KUKA KRL program: EPS_2_25862_MH01_A_20251016040654.src

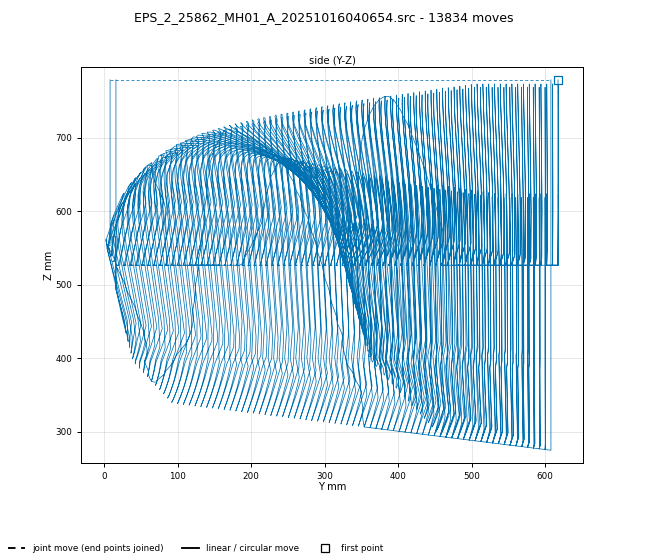
[picture p0: tool path of EPS_2_25862_MH01_A_20251016040654.src, 13834 of 13836 moves have a stored position in this frame; points joined in program order, loops and branches not executed]
&ACCESS RVP
&REL 4
&COMMENT QRS 19112012
&PARAM EDITMASK = *
DEF PART()
EXT BAS (BAS_COMMAND :IN,REAL :IN )
INT I
BAS (#INITMOV,0 )

;KUKA QRS Post kuka4.cps  Date:22-06-2017 !

File_ID=2893

QRS_PRE_INIT()

;Init var - Until changes are made in qrs_pre_init
Outlet_Square_prg=0
Inlet_1_Square_prg=0
Inlet_2_Square_prg=0
Inlet_3_Square_prg=0
Inlet_4_Square_prg=0
Inlet_5_Square_prg=0

Outlet_1={X 0.000, Y 506.950, Z 586.000, B 0.000, E1 0.000 }
Inlet_1={X 0.000, Y 532.640, Z 498.500, B 0.000, E1 270.000 }
Outlet_1_type=366
Inlet_1_type=201
;QRS#1=Sidecore dimensions
;QRS#2=375-15" PVC SDR 35
;QRS#3=200-8" PVC SDR 35
;QRS#4=
;QRS#5=
;QRS#6=
;QRS#7=
;QRS#8=
;QRS#9=20Y PSX
;QRS#10=12-08 PSX
;QRS#11=
;QRS#12=
;QRS#13=
;QRS#14=
;QRS#15=
;QRS#16=1220x127x1067 3,5'
;QRS#17=EPS Height
;QRS#18=769
;QRS#19=*
;QRS#20= UPDATED VERSION 22-06-2017
;QRS#21=*
Outlet_Square=0250
Inlet_1_Square=0100
Inlet_2_Square=0
Inlet_3_Square=0
Inlet_4_Square=0
Inlet_5_Square=0
Mill_Square=1
Outlet_Square_Prg=252
Inlet_1_Square_prg=204

QRS_INIT()

$ADVANCE=5

; T1
PTP {E1 171.211,E2 171.211}
PTP {X 0,Y 617.567,A -85,B 0,C 180,E1 171.211,E2 171.211,E3 0,E4 0,E5 0,E6 0}
QRS_SPEED_INIT()
LIN {X 0,Y 617.567,Z 779,A -85,B 0,C 180,E1 171.211,E2 171.211,E3 0,E4 0,E5 0,E6 0} C_VEL
LIN {X 0,Y 617.567,Z 528.81,A -85,B 0,C 180,E1 171.211,E2 171.211} C_VEL
LIN {X 0,Y 617.544,Z 526.81,A -85,B 0,C 180,E1 171.397,E2 171.397} C_VEL
LIN {X 0,Y 617.991,Z 526.81,A -85,B 0,C 180,E1 174.215,E2 174.215} C_VEL
LIN {X 0,Y 618.006,Z 526.81,A -85,B 0,C 180,E1 178.846,E2 178.846} C_VEL
LIN {X 0,Y 618.053,Z 526.81,A -85,B 0,C 180,E1 183.469,E2 183.469} C_VEL
LIN {X 0,Y 617.988,Z 526.81,A -85,B 0,C 180,E1 188.116,E2 188.116} C_VEL
LIN {X 0,Y 617.951,Z 526.81,A -85,B 0,C 180,E1 192.817,E2 192.817} C_VEL
LIN {X 0,Y 617.958,Z 526.81,A -85,B 0,C 180,E1 197.608,E2 197.608} C_VEL
LIN {X 0,Y 617.766,Z 526.81,A -85,B 0,C 180,E1 198.549,E2 198.549} C_VEL
LIN {X 0,Y 617.884,Z 526.81,A -85,B 0,C 180,E1 202.532,E2 202.532} C_VEL
LIN {X 0,Y 617.406,Z 526.81,A -85,B 0,C 180,E1 205.079,E2 205.079} C_VEL
LIN {X 0,Y 617.875,Z 526.81,A -85,B 0,C 180,E1 207.638,E2 207.638} C_VEL
LIN {X 0,Y 617.419,Z 526.81,A -85,B 0,C 180,E1 210.304,E2 210.304} C_VEL
LIN {X 0,Y 617.937,Z 526.81,A -85,B 0,C 180,E1 212.99,E2 212.99} C_VEL
LIN {X 0,Y 617.675,Z 526.81,A -85,B 0,C 180,E1 215.809,E2 215.809} C_VEL
LIN {X 0,Y 617.669,Z 526.81,A -85,B 0,C 180,E1 218.112,E2 218.112} C_VEL
LIN {X 0,Y 617.756,Z 526.81,A -85,B 0,C 180,E1 221.735,E2 221.735} C_VEL
LIN {X 0,Y 617.383,Z 526.81,A -85,B 0,C 180,E1 225.055,E2 225.055} C_VEL
LIN {X 0,Y 617.751,Z 526.81,A -85,B 0,C 180,E1 228.278,E2 228.278} C_VEL
LIN {X 0,Y 617.353,Z 526.81,A -85,B 0,C 180,E1 231.927,E2 231.927} C_VEL
LIN {X 0,Y 617.814,Z 526.81,A -85,B 0,C 180,E1 234.203,E2 234.203} C_VEL
LIN {X 0,Y 617.316,Z 526.81,A -85,B 0,C 180,E1 236.974,E2 236.974} C_VEL
LIN {X 0,Y 617.844,Z 526.81,A -85,B 0,C 180,E1 239.721,E2 239.721} C_VEL
LIN {X 0,Y 617.407,Z 526.81,A -85,B 0,C 180,E1 242.341,E2 242.341} C_VEL
LIN {X 0,Y 617.943,Z 526.81,A -85,B 0,C 180,E1 244.946,E2 244.946} C_VEL
LIN {X 0,Y 618.003,Z 526.81,A -85,B 0,C 180,E1 249.132,E2 249.132} C_VEL
LIN {X 0,Y 617.672,Z 526.81,A -85,B 0,C 180,E1 249.232,E2 249.232} C_VEL
LIN {X 0,Y 617.573,Z 527.124,A -85,B 0,C 180,E1 249.254,E2 249.254} C_VEL
LIN {X 0,Y 617.998,Z 591.592,A -85,B 0,C 180,E1 250.062,E2 250.062} C_VEL
LIN {X 0,Y 618.002,Z 600.715,A -85,B 0,C 180,E1 250.212,E2 250.212} C_VEL
LIN {X 0,Y 617.91,Z 609.031,A -85,B 0,C 180,E1 250.381,E2 250.381} C_VEL
LIN {X 0,Y 617.97,Z 618.416,A -85,B 0,C 180,E1 250.619,E2 250.619} C_VEL
LIN {X 0,Y 617.998,Z 627.724,A -85,B 0,C 180,E1 250.899,E2 250.899} C_VEL
LIN {X 0,Y 617.96,Z 636.377,A -85,B 0,C 180,E1 251.197,E2 251.197} C_VEL
LIN {X 0,Y 617.966,Z 645.125,A -85,B 0,C 180,E1 251.542,E2 251.542} C_VEL
LIN {X 0,Y 618.001,Z 654.313,A -85,B 0,C 180,E1 251.955,E2 251.955} C_VEL
LIN {X 0,Y 617.987,Z 663.052,A -85,B 0,C 180,E1 252.395,E2 252.395} C_VEL
LIN {X 0,Y 617.974,Z 670.423,A -85,B 0,C 180,E1 252.803,E2 252.803} C_VEL
LIN {X 0,Y 617.99,Z 678.723,A -85,B 0,C 180,E1 253.313,E2 253.313} C_VEL
LIN {X 0,Y 617.989,Z 687.493,A -85,B 0,C 180,E1 253.911,E2 253.911} C_VEL
LIN {X 0,Y 617.973,Z 695.458,A -85,B 0,C 180,E1 254.511,E2 254.511} C_VEL
LIN {X 0,Y 617.955,Z 702.634,A -85,B 0,C 180,E1 255.102,E2 255.102} C_VEL
LIN {X 0,Y 617.942,Z 709.277,A -85,B 0,C 180,E1 255.699,E2 255.699} C_VEL
LIN {X 0,Y 617.983,Z 715.369,A -85,B 0,C 180,E1 256.295,E2 256.295} C_VEL
LIN {X 0,Y 617.985,Z 720.995,A -85,B 0,C 180,E1 256.889,E2 256.889} C_VEL
LIN {X 0,Y 617.92,Z 727.418,A -85,B 0,C 180,E1 257.628,E2 257.628} C_VEL
LIN {X 0,Y 617.926,Z 733.244,A -85,B 0,C 180,E1 258.366,E2 258.366} C_VEL
LIN {X 0,Y 617.973,Z 737.547,A -85,B 0,C 180,E1 258.956,E2 258.956} C_VEL
LIN {X 0,Y 617.979,Z 742.76,A -85,B 0,C 180,E1 259.742,E2 259.742} C_VEL
LIN {X 0,Y 617.882,Z 748.578,A -85,B 0,C 180,E1 260.724,E2 260.724} C_VEL
LIN {X 0,Y 617.911,Z 752.668,A -85,B 0,C 180,E1 261.501,E2 261.501} C_VEL
LIN {X 0,Y 618.002,Z 756.64,A -85,B 0,C 180,E1 262.353,E2 262.353} C_VEL
LIN {X 0,Y 617.904,Z 760.475,A -85,B 0,C 180,E1 263.283,E2 263.283} C_VEL
LIN {X 0,Y 617.879,Z 762.222,A -85,B 0,C 180,E1 263.748,E2 263.748} C_VEL
LIN {X 0,Y 617.937,Z 765.214,A -85,B 0,C 180,E1 264.678,E2 264.678} C_VEL
LIN {X 0,Y 617.962,Z 767.691,A -85,B 0,C 180,E1 265.606,E2 265.606} C_VEL
LIN {X 0,Y 617.845,Z 769.703,A -85,B 0,C 180,E1 266.532,E2 266.532} C_VEL
LIN {X 0,Y 617.849,Z 771.199,A -85,B 0,C 180,E1 267.457,E2 267.457} C_VEL
LIN {X 0,Y 617.951,Z 772.526,A -85,B 0,C 180,E1 268.845,E2 268.845} C_VEL
LIN {X 0,Y 617.842,Z 772.907,A -85,B 0,C 180,E1 269.769,E2 269.769} C_VEL
LIN {X 0,Y 617.828,Z 772.91,A -85,B 0,C 180,E1 270.232,E2 270.232} C_VEL
LIN {X 0,Y 617.89,Z 772.542,A -85,B 0,C 180,E1 271.156,E2 271.156} C_VEL
LIN {X 0,Y 617.878,Z 771.19,A -85,B 0,C 180,E1 272.544,E2 272.544} C_VEL
LIN {X 0,Y 617.83,Z 769.706,A -85,B 0,C 180,E1 273.47,E2 273.47} C_VEL
LIN {X 0,Y 617.92,Z 767.699,A -85,B 0,C 180,E1 274.396,E2 274.396} C_VEL
LIN {X 0,Y 617.979,Z 765.199,A -85,B 0,C 180,E1 275.323,E2 275.323} C_VEL
LIN {X 0,Y 617.884,Z 762.216,A -85,B 0,C 180,E1 276.253,E2 276.253} C_VEL
LIN {X 0,Y 617.945,Z 757.648,A -85,B 0,C 180,E1 277.416,E2 277.416} C_VEL
LIN {X 0,Y 617.97,Z 754.519,A -85,B 0,C 180,E1 278.115,E2 278.115} C_VEL
LIN {X 0,Y 617.888,Z 749.593,A -85,B 0,C 180,E1 279.09,E2 279.09} C_VEL
LIN {X 0,Y 617.902,Z 745.133,A -85,B 0,C 180,E1 279.871,E2 279.871} C_VEL
LIN {X 0,Y 617.972,Z 741.485,A -85,B 0,C 180,E1 280.457,E2 280.457} C_VEL
LIN {X 0,Y 617.979,Z 735.404,A -85,B 0,C 180,E1 281.339,E2 281.339} C_VEL
LIN {X 0,Y 617.924,Z 729.803,A -85,B 0,C 180,E1 282.078,E2 282.078} C_VEL
LIN {X 0,Y 617.94,Z 723.617,A -85,B 0,C 180,E1 282.817,E2 282.817} C_VEL
LIN {X 0,Y 618.001,Z 718.223,A -85,B 0,C 180,E1 283.409,E2 283.409} C_VEL
LIN {X 0,Y 617.984,Z 710.825,A -85,B 0,C 180,E1 284.152,E2 284.152} C_VEL
LIN {X 0,Y 617.966,Z 704.331,A -85,B 0,C 180,E1 284.749,E2 284.749} C_VEL
LIN {X 0,Y 617.984,Z 696.644,A -85,B 0,C 180,E1 285.394,E2 285.394} C_VEL
LIN {X 0,Y 617.986,Z 690.265,A -85,B 0,C 180,E1 285.886,E2 285.886} C_VEL
LIN {X 0,Y 618,Z 681.693,A -85,B 0,C 180,E1 286.489,E2 286.489} C_VEL
LIN {X 0,Y 617.987,Z 673.739,A -85,B 0,C 180,E1 286.996,E2 286.996} C_VEL
LIN {X 0,Y 617.97,Z 664.896,A -85,B 0,C 180,E1 287.505,E2 287.505} C_VEL
LIN {X 0,Y 617.953,Z 657.854,A -85,B 0,C 180,E1 287.873,E2 287.873} C_VEL
LIN {X 0,Y 617.995,Z 649.403,A -85,B 0,C 180,E1 288.27,E2 288.27} C_VEL
LIN {X 0,Y 617.999,Z 641.397,A -85,B 0,C 180,E1 288.609,E2 288.609} C_VEL
LIN {X 0,Y 617.905,Z 631.678,A -85,B 0,C 180,E1 288.973,E2 288.973} C_VEL
LIN {X 0,Y 618.012,Z 622.258,A -85,B 0,C 180,E1 289.27,E2 289.27} C_VEL
LIN {X 0,Y 618.03,Z 612.701,A -85,B 0,C 180,E1 289.528,E2 289.528} C_VEL
LIN {X 0,Y 617.968,Z 602.985,A -85,B 0,C 180,E1 289.746,E2 289.746} C_VEL
LIN {X 0,Y 617.848,Z 594.545,A -85,B 0,C 180,E1 289.901,E2 289.901} C_VEL
LIN {X 0,Y 617.823,Z 577.609,A -85,B 0,C 180,E1 290.124,E2 290.124} C_VEL
LIN {X 0,Y 617.563,Z 526.827,A -85,B 0,C 180,E1 290.75,E2 290.75} C_VEL
LIN {X 0,Y 618.055,Z 526.81,A -85,B 0,C 180,E1 290.891,E2 290.891} C_VEL
LIN {X 0,Y 617.945,Z 526.81,A -85,B 0,C 180,E1 295.055,E2 295.055} C_VEL
LIN {X 0,Y 617.401,Z 526.81,A -85,B 0,C 180,E1 297.66,E2 297.66} C_VEL
LIN {X 0,Y 617.83,Z 526.81,A -85,B 0,C 180,E1 300.281,E2 300.281} C_VEL
LIN {X 0,Y 617.31,Z 526.81,A -85,B 0,C 180,E1 303.028,E2 303.028} C_VEL
LIN {X 0,Y 617.818,Z 526.81,A -85,B 0,C 180,E1 305.798,E2 305.798} C_VEL
LIN {X 0,Y 617.553,Z 526.81,A -85,B 0,C 180,E1 308.722,E2 308.722} C_VEL
LIN {X 0,Y 617.772,Z 526.81,A -85,B 0,C 180,E1 311.733,E2 311.733} C_VEL
LIN {X 0,Y 617.89,Z 526.81,A -85,B 0,C 180,E1 315.1,E2 315.1} C_VEL
LIN {X 0,Y 617.463,Z 526.81,A -85,B 0,C 180,E1 318.307,E2 318.307} C_VEL
LIN {X 0,Y 617.793,Z 526.81,A -85,B 0,C 180,E1 321.295,E2 321.295} C_VEL
LIN {X 0,Y 617.729,Z 526.81,A -85,B 0,C 180,E1 325.801,E2 325.801} C_VEL
LIN {X 0,Y 617.882,Z 526.81,A -85,B 0,C 180,E1 327.006,E2 327.006} C_VEL
LIN {X 0,Y 617.635,Z 526.81,A -85,B 0,C 180,E1 330.177,E2 330.177} C_VEL
LIN {X 0,Y 617.646,Z 526.81,A -85,B 0,C 180,E1 332.351,E2 332.351} C_VEL
LIN {X 0,Y 617.512,Z 526.81,A -85,B 0,C 180,E1 335.244,E2 335.244} C_VEL
LIN {X 0,Y 617.731,Z 526.81,A -85,B 0,C 180,E1 337.462,E2 337.462} C_VEL
LIN {X 0,Y 617.771,Z 526.81,A -85,B 0,C 180,E1 341.453,E2 341.453} C_VEL
LIN {X 0,Y 617.968,Z 526.81,A -85,B 0,C 180,E1 342.392,E2 342.392} C_VEL
LIN {X 0,Y 617.72,Z 526.81,A -85,B 0,C 180,E1 347.178,E2 347.178} C_VEL
LIN {X 0,Y 617.945,Z 526.81,A -85,B 0,C 180,E1 348.034,E2 348.034} C_VEL
LIN {X 0,Y 617.433,Z 526.895,A -85,B 0,C 180,E1 348.173,E2 348.173} C_VEL
LIN {X 0,Y 617.979,Z 531.008,A -85,B 0,C 180,E1 348.301,E2 348.301} C_VEL
LIN {X 0,Y 617.99,Z 539.274,A -85,B 0,C 180,E1 348.568,E2 348.568} C_VEL
LIN {X 0,Y 618.035,Z 547.303,A -85,B 0,C 180,E1 348.887,E2 348.887} C_VEL
LIN {X 0,Y 618.042,Z 554.943,A -85,B 0,C 180,E1 349.245,E2 349.245} C_VEL
LIN {X 0,Y 617.989,Z 563.583,A -85,B 0,C 180,E1 349.726,E2 349.726} C_VEL
LIN {X 0,Y 618.017,Z 570.585,A -85,B 0,C 180,E1 350.186,E2 350.186} C_VEL
LIN {X 0,Y 618.022,Z 577.883,A -85,B 0,C 180,E1 350.735,E2 350.735} C_VEL
LIN {X 0,Y 617.995,Z 584.768,A -85,B 0,C 180,E1 351.337,E2 351.337} C_VEL
LIN {X 0,Y 617.992,Z 591.346,A -85,B 0,C 180,E1 352.001,E2 352.001} C_VEL
LIN {X 0,Y 617.99,Z 596.368,A -85,B 0,C 180,E1 352.584,E2 352.584} C_VEL
LIN {X 0,Y 617.999,Z 601.64,A -85,B 0,C 180,E1 353.282,E2 353.282} C_VEL
LIN {X 0,Y 617.979,Z 606.155,A -85,B 0,C 180,E1 353.98,E2 353.98} C_VEL
LIN {X 0,Y 617.965,Z 610.06,A -85,B 0,C 180,E1 354.676,E2 354.676} C_VEL
LIN {X 0,Y 618.005,Z 613.315,A -85,B 0,C 180,E1 355.372,E2 355.372} C_VEL
LIN {X 0,Y 617.99,Z 616.083,A -85,B 0,C 180,E1 356.067,E2 356.067} C_VEL
LIN {X 0,Y 617.961,Z 617.642,A -85,B 0,C 180,E1 356.53,E2 356.53} C_VEL
LIN {X 0,Y 617.962,Z 618.985,A -85,B 0,C 180,E1 356.993,E2 356.993} C_VEL
LIN {X 0,Y 617.986,Z 620.121,A -85,B 0,C 180,E1 357.456,E2 357.456} C_VEL
LIN {X 0,Y 617.984,Z 621.822,A -85,B 0,C 180,E1 358.381,E2 358.381} C_VEL
LIN {X 0,Y 617.941,Z 622.381,A -85,B 0,C 180,E1 358.843,E2 358.843} C_VEL
LIN {X 0,Y 617.943,Z 622.891,A -85,B 0,C 180,E1 359.767,E2 359.767} C_VEL
LIN {X 0,Y 617.998,Z 622.65,A -85,B 0,C 180,E1 360.692,E2 360.692} C_VEL
LIN {X 0,Y 617.929,Z 621.709,A -85,B 0,C 180,E1 361.616,E2 361.616} C_VEL
LIN {X 0,Y 617.952,Z 619.943,A -85,B 0,C 180,E1 362.541,E2 362.541} C_VEL
LIN {X 0,Y 617.986,Z 617.357,A -85,B 0,C 180,E1 363.467,E2 363.467} C_VEL
LIN {X 0,Y 617.958,Z 615.767,A -85,B 0,C 180,E1 363.93,E2 363.93} C_VEL
LIN {X 0,Y 617.962,Z 612.953,A -85,B 0,C 180,E1 364.625,E2 364.625} C_VEL
LIN {X 0,Y 618.012,Z 609.592,A -85,B 0,C 180,E1 365.32,E2 365.32} C_VEL
LIN {X 0,Y 618.005,Z 605.617,A -85,B 0,C 180,E1 366.017,E2 366.017} C_VEL
LIN {X 0,Y 617.996,Z 601.043,A -85,B 0,C 180,E1 366.715,E2 366.715} C_VEL
LIN {X 0,Y 618.007,Z 595.651,A -85,B 0,C 180,E1 367.413,E2 367.413} C_VEL
LIN {X 0,Y 618.016,Z 589.425,A -85,B 0,C 180,E1 368.112,E2 368.112} C_VEL
LIN {X 0,Y 618.01,Z 582.569,A -85,B 0,C 180,E1 368.777,E2 368.777} C_VEL
LIN {X 0,Y 617.987,Z 575.788,A -85,B 0,C 180,E1 369.34,E2 369.34} C_VEL
LIN {X 0,Y 618.031,Z 568.063,A -85,B 0,C 180,E1 369.896,E2 369.896} C_VEL
LIN {X 0,Y 618.031,Z 560.563,A -85,B 0,C 180,E1 370.36,E2 370.36} C_VEL
LIN {X 0,Y 617.996,Z 552.876,A -85,B 0,C 180,E1 370.768,E2 370.768} C_VEL
LIN {X 0,Y 618.051,Z 545.241,A -85,B 0,C 180,E1 371.11,E2 371.11} C_VEL
LIN {X 0,Y 618.043,Z 537.066,A -85,B 0,C 180,E1 371.418,E2 371.418} C_VEL
LIN {X 0,Y 617.95,Z 527.367,A -85,B 0,C 180,E1 371.71,E2 371.71} C_VEL
LIN {X 0,Y 617.836,Z 526.81,A -85,B 0,C 180,E1 371.732,E2 371.732} C_VEL
LIN {X 0,Y 618.049,Z 526.81,A -85,B 0,C 180,E1 371.961,E2 371.961} C_VEL
LIN {X 0,Y 617.965,Z 526.81,A -85,B 0,C 180,E1 377.604,E2 377.604} C_VEL
LIN {X 0,Y 617.784,Z 526.81,A -85,B 0,C 180,E1 378.551,E2 378.551} C_VEL
LIN {X 0,Y 617.94,Z 526.81,A -85,B 0,C 180,E1 382.527,E2 382.527} C_VEL
LIN {X 0,Y 617.438,Z 526.81,A -85,B 0,C 180,E1 385.074,E2 385.074} C_VEL
LIN {X 0,Y 617.879,Z 526.81,A -85,B 0,C 180,E1 387.634,E2 387.634} C_VEL
LIN {X 0,Y 617.37,Z 526.81,A -85,B 0,C 180,E1 390.303,E2 390.303} C_VEL
LIN {X 0,Y 617.844,Z 526.81,A -85,B 0,C 180,E1 392.992,E2 392.992} C_VEL
LIN {X 0,Y 617.702,Z 526.81,A -85,B 0,C 180,E1 394.195,E2 394.195} C_VEL
LIN {X 0,Y 617.786,Z 526.81,A -85,B 0,C 180,E1 398.701,E2 398.701} C_VEL
LIN {X 0,Y 617.438,Z 526.81,A -85,B 0,C 180,E1 401.757,E2 401.757} C_VEL
LIN {X 0,Y 617.869,Z 526.81,A -85,B 0,C 180,E1 404.898,E2 404.898} C_VEL
LIN {X 0,Y 617.794,Z 526.81,A -85,B 0,C 180,E1 408.269,E2 408.269} C_VEL
LIN {X 0,Y 617.56,Z 526.81,A -85,B 0,C 180,E1 411.279,E2 411.279} C_VEL
LIN {X 0,Y 617.58,Z 526.81,A -85,B 0,C 180,E1 411.896,E2 411.896} C_VEL
LIN {X 0,Y 617.811,Z 526.81,A -85,B 0,C 180,E1 414.201,E2 414.201} C_VEL
LIN {X 0,Y 617.354,Z 526.81,A -85,B 0,C 180,E1 416.975,E2 416.975} C_VEL
LIN {X 0,Y 617.897,Z 526.81,A -85,B 0,C 180,E1 419.722,E2 419.722} C_VEL
LIN {X 0,Y 617.42,Z 526.81,A -85,B 0,C 180,E1 422.341,E2 422.341} C_VEL
LIN {X 0,Y 617.901,Z 526.81,A -85,B 0,C 180,E1 424.943,E2 424.943} C_VEL
LIN {X 0,Y 617.445,Z 526.81,A -85,B 0,C 180,E1 427.451,E2 427.451} C_VEL
LIN {X 0,Y 617.945,Z 526.81,A -85,B 0,C 180,E1 429.951,E2 429.951} C_VEL
LIN {X 0,Y 618.027,Z 526.81,A -85,B 0,C 180,E1 433.628,E2 433.628} C_VEL
LIN {X 0,Y 618.006,Z 526.81,A -85,B 0,C 180,E1 439.544,E2 439.544} C_VEL
LIN {X 0,Y 618.005,Z 526.81,A -85,B 0,C 180,E1 444.213,E2 444.213} C_VEL
LIN {X 0,Y 618.056,Z 526.81,A -85,B 0,C 180,E1 448.844,E2 448.844} C_VEL
LIN {X 0,Y 618.059,Z 526.81,A -85,B 0,C 180,E1 453.467,E2 453.467} C_VEL
LIN {X 0,Y 617.996,Z 526.81,A -85,B 0,C 180,E1 458.114,E2 458.114} C_VEL
LIN {X 0,Y 618.005,Z 526.81,A -85,B 0,C 180,E1 462.814,E2 462.814} C_VEL
LIN {X 0,Y 617.945,Z 526.81,A -85,B 0,C 180,E1 467.606,E2 467.606} C_VEL
LIN {X 0,Y 617.762,Z 526.81,A -85,B 0,C 180,E1 468.554,E2 468.554} C_VEL
LIN {X 0,Y 617.921,Z 526.81,A -85,B 0,C 180,E1 472.529,E2 472.529} C_VEL
LIN {X 0,Y 617.422,Z 526.81,A -85,B 0,C 180,E1 475.076,E2 475.076} C_VEL
LIN {X 0,Y 617.864,Z 526.81,A -85,B 0,C 180,E1 477.637,E2 477.637} C_VEL
LIN {X 0,Y 617.365,Z 526.81,A -85,B 0,C 180,E1 480.305,E2 480.305} C_VEL
LIN {X 0,Y 617.849,Z 526.81,A -85,B 0,C 180,E1 482.994,E2 482.994} C_VEL
LIN {X 0,Y 617.717,Z 526.81,A -85,B 0,C 180,E1 484.202,E2 484.202} C_VEL
LIN {X 0,Y 617.776,Z 526.81,A -85,B 0,C 180,E1 488.704,E2 488.704} C_VEL
LIN {X 0,Y 617.417,Z 526.81,A -85,B 0,C 180,E1 491.761,E2 491.761} C_VEL
LIN {X 0,Y 617.82,Z 526.81,A -85,B 0,C 180,E1 494.905,E2 494.905} C_VEL
LIN {X 0,Y 617.766,Z 526.81,A -85,B 0,C 180,E1 498.274,E2 498.274} C_VEL
LIN {X 0,Y 617.556,Z 526.81,A -85,B 0,C 180,E1 501.282,E2 501.282} C_VEL
LIN {X 0,Y 617.832,Z 526.81,A -85,B 0,C 180,E1 504.206,E2 504.206} C_VEL
LIN {X 0,Y 617.356,Z 526.81,A -85,B 0,C 180,E1 506.978,E2 506.978} C_VEL
LIN {X 0,Y 617.899,Z 526.81,A -85,B 0,C 180,E1 509.725,E2 509.725} C_VEL
LIN {X 0,Y 617.405,Z 526.81,A -85,B 0,C 180,E1 512.343,E2 512.343} C_VEL
LIN {X 0,Y 617.874,Z 526.81,A -85,B 0,C 180,E1 514.945,E2 514.945} C_VEL
LIN {X 0,Y 617.444,Z 526.81,A -85,B 0,C 180,E1 517.454,E2 517.454} C_VEL
LIN {X 0,Y 617.969,Z 526.81,A -85,B 0,C 180,E1 519.954,E2 519.954} C_VEL
LIN {X 0,Y 618.057,Z 526.81,A -85,B 0,C 180,E1 523.625,E2 523.625} C_VEL
LIN {X 0,Y 618.006,Z 526.81,A -85,B 0,C 180,E1 529.546,E2 529.546} C_VEL
LIN {X 0,Y 617.544,Z 526.81,A -85,B 0,C 180,E1 531.397,E2 531.397} C_VEL
LIN {X 0,Y 613.845,Z 526.81,A -85,B 0,C 180,E1 532.988,E2 532.988} C_VEL
LIN {X 0,Y 609.944,Z 526.81,A -85,B 0,C 180,E1 534.598,E2 534.598} C_VEL
LIN {X 0,Y 609.767,Z 526.81,A -85,B 0,C 180,E1 539.996,E2 539.996} C_VEL
LIN {X 0,Y 609.877,Z 526.81,A -85,B 0,C 180,E1 544.267,E2 544.267} C_VEL
LIN {X 0,Y 609.912,Z 526.81,A -85,B 0,C 180,E1 548.561,E2 548.561} C_VEL
LIN {X 0,Y 610.024,Z 526.81,A -85,B 0,C 180,E1 552.902,E2 552.902} C_VEL
LIN {X 0,Y 609.801,Z 526.81,A -85,B 0,C 180,E1 558.825,E2 558.825} C_VEL
LIN {X 0,Y 609.689,Z 526.81,A -85,B 0,C 180,E1 563.406,E2 563.406} C_VEL
LIN {X 0,Y 609.802,Z 526.81,A -85,B 0,C 180,E1 568.141,E2 568.141} C_VEL
LIN {X 0,Y 610.014,Z 526.81,A -85,B 0,C 180,E1 573.089,E2 573.089} C_VEL
LIN {X 0,Y 609.701,Z 526.81,A -85,B 0,C 180,E1 578.368,E2 578.368} C_VEL
LIN {X 0,Y 609.712,Z 526.81,A -85,B 0,C 180,E1 582.095,E2 582.095} C_VEL
LIN {X 0,Y 609.791,Z 526.81,A -85,B 0,C 180,E1 588.139,E2 588.139} C_VEL
LIN {X 0,Y 609.673,Z 526.81,A -85,B 0,C 180,E1 593.419,E2 593.419} C_VEL
LIN {X 0,Y 609.781,Z 526.81,A -85,B 0,C 180,E1 600.229,E2 600.229} C_VEL
LIN {X 0,Y 610.026,Z 526.81,A -85,B 0,C 180,E1 605.047,E2 605.047} C_VEL
LIN {X 0,Y 610.064,Z 526.839,A -85,B 0,C 180,E1 608.983,E2 608.983} C_VEL
LIN {X 0,Y 610.516,Z 606.691,A -85,B 0,C 180,E1 610.077,E2 610.077} C_VEL
LIN {X 0,Y 610.436,Z 640.436,A -85,B 0,C 180,E1 611.114,E2 611.114} C_VEL
LIN {X 0,Y 610.334,Z 672.149,A -85,B 0,C 180,E1 612.685,E2 612.685} C_VEL
LIN {X 0,Y 610.259,Z 700.151,A -85,B 0,C 180,E1 614.678,E2 614.678} C_VEL
LIN {X 0,Y 610.211,Z 724.689,A -85,B 0,C 180,E1 617.1,E2 617.1} C_VEL
LIN {X 0,Y 610.176,Z 744.633,A -85,B 0,C 180,E1 619.82,E2 619.82} C_VEL
LIN {X 0,Y 610.138,Z 760.105,A -85,B 0,C 180,E1 622.876,E2 622.876} C_VEL
LIN {X 0,Y 610.138,Z 769.078,A -85,B 0,C 180,E1 625.734,E2 625.734} C_VEL
LIN {X 0,Y 610.097,Z 773.418,A -85,B 0,C 180,E1 628.581,E2 628.581} C_VEL
LIN {X 0,Y 610.054,Z 773.413,A -85,B 0,C 180,E1 631.426,E2 631.426} C_VEL
LIN {X 0,Y 610.083,Z 769.063,A -85,B 0,C 180,E1 634.273,E2 634.273} C_VEL
LIN {X 0,Y 610.151,Z 758.546,A -85,B 0,C 180,E1 637.489,E2 637.489} C_VEL
LIN {X 0,Y 610.185,Z 742.34,A -85,B 0,C 180,E1 640.548,E2 640.548} C_VEL
LIN {X 0,Y 610.211,Z 721.418,A -85,B 0,C 180,E1 643.272,E2 643.272} C_VEL
LIN {X 0,Y 610.288,Z 695.834,A -85,B 0,C 180,E1 645.67,E2 645.67} C_VEL
LIN {X 0,Y 610.359,Z 667.256,A -85,B 0,C 180,E1 647.601,E2 647.601} C_VEL
LIN {X 0,Y 610.454,Z 634.794,A -85,B 0,C 180,E1 649.105,E2 649.105} C_VEL
LIN {X 0,Y 610.49,Z 600.135,A -85,B 0,C 180,E1 650.053,E2 650.053} C_VEL
LIN {X 0,Y 610.11,Z 526.81,A -85,B 0,C 180,E1 651.046,E2 651.046} C_VEL
LIN {X 0,Y 610.033,Z 526.81,A -85,B 0,C 180,E1 654.96,E2 654.96} C_VEL
LIN {X 0,Y 609.762,Z 526.81,A -85,B 0,C 180,E1 659.78,E2 659.78} C_VEL
LIN {X 0,Y 609.718,Z 526.81,A -85,B 0,C 180,E1 666.586,E2 666.586} C_VEL
LIN {X 0,Y 609.78,Z 526.81,A -85,B 0,C 180,E1 672.103,E2 672.103} C_VEL
LIN {X 0,Y 609.523,Z 526.81,A -85,B 0,C 180,E1 677.889,E2 677.889} C_VEL
LIN {X 0,Y 609.488,Z 526.81,A -85,B 0,C 180,E1 682.654,E2 682.654} C_VEL
LIN {X 0,Y 609.824,Z 526.81,A -85,B 0,C 180,E1 687.587,E2 687.587} C_VEL
LIN {X 0,Y 609.683,Z 526.81,A -85,B 0,C 180,E1 691.853,E2 691.853} C_VEL
LIN {X 0,Y 609.663,Z 526.81,A -85,B 0,C 180,E1 696.771,E2 696.771} C_VEL
LIN {X 0,Y 609.947,Z 526.81,A -85,B 0,C 180,E1 702.675,E2 702.675} C_VEL
LIN {X 0,Y 609.764,Z 526.81,A -85,B 0,C 180,E1 708.003,E2 708.003} C_VEL
LIN {X 0,Y 610.311,Z 553.498,A -85,B 0,C 180,E1 709.011,E2 709.011} C_VEL
LIN {X 0,Y 610.246,Z 576.43,A -85,B 0,C 180,E1 710.454,E2 710.454} C_VEL
LIN {X 0,Y 610.193,Z 595.738,A -85,B 0,C 180,E1 712.32,E2 712.32} C_VEL
LIN {X 0,Y 610.161,Z 609.339,A -85,B 0,C 180,E1 714.308,E2 714.308} C_VEL
LIN {X 0,Y 610.141,Z 619.6,A -85,B 0,C 180,E1 716.804,E2 716.804} C_VEL
LIN {X 0,Y 610.148,Z 623.152,A -85,B 0,C 180,E1 718.583,E2 718.583} C_VEL
LIN {X 0,Y 610.156,Z 623.995,A -85,B 0,C 180,E1 720.004,E2 720.004} C_VEL
LIN {X 0,Y 610.126,Z 621.914,A -85,B 0,C 180,E1 722.138,E2 722.138} C_VEL
LIN {X 0,Y 610.157,Z 614.128,A -85,B 0,C 180,E1 724.63,E2 724.63} C_VEL
LIN {X 0,Y 610.19,Z 600.493,A -85,B 0,C 180,E1 726.984,E2 726.984} C_VEL
LIN {X 0,Y 610.231,Z 581.767,A -85,B 0,C 180,E1 729.015,E2 729.015} C_VEL
LIN {X 0,Y 610.277,Z 560.182,A -85,B 0,C 180,E1 730.547,E2 730.547} C_VEL
LIN {X 0,Y 610.312,Z 534.106,A -85,B 0,C 180,E1 731.678,E2 731.678} C_VEL
LIN {X 0,Y 610.071,Z 526.81,A -85,B 0,C 180,E1 731.909,E2 731.909} C_VEL
LIN {X 0,Y 609.946,Z 526.81,A -85,B 0,C 180,E1 737.334,E2 737.334} C_VEL
LIN {X 0,Y 609.744,Z 526.81,A -85,B 0,C 180,E1 743.413,E2 743.413} C_VEL
LIN {X 0,Y 609.784,Z 526.81,A -85,B 0,C 180,E1 748.152,E2 748.152} C_VEL
LIN {X 0,Y 609.924,Z 526.81,A -85,B 0,C 180,E1 753.105,E2 753.105} C_VEL
LIN {X 0,Y 609.59,Z 526.81,A -85,B 0,C 180,E1 759.644,E2 759.644} C_VEL
LIN {X 0,Y 609.721,Z 526.81,A -85,B 0,C 180,E1 765.944,E2 765.944} C_VEL
LIN {X 0,Y 609.551,Z 526.81,A -85,B 0,C 180,E1 770.358,E2 770.358} C_VEL
LIN {X 0,Y 609.61,Z 526.81,A -85,B 0,C 180,E1 775.159,E2 775.159} C_VEL
LIN {X 0,Y 609.782,Z 526.81,A -85,B 0,C 180,E1 780.351,E2 780.351} C_VEL
LIN {X 0,Y 609.978,Z 526.81,A -85,B 0,C 180,E1 785.037,E2 785.037} C_VEL
LIN {X 0,Y 609.794,Z 526.81,A -85,B 0,C 180,E1 791.165,E2 791.165} C_VEL
LIN {X 0,Y 609.369,Z 526.81,A -85,B 0,C 180,E1 795.705,E2 795.705} C_VEL
LIN {X 0,Y 609.937,Z 526.81,A -85,B 0,C 180,E1 799.99,E2 799.99} C_VEL
LIN {X 0,Y 610.087,Z 526.81,A -85,B 0,C 180,E1 804.3,E2 804.3} C_VEL
LIN {X 0,Y 609.785,Z 526.81,A -85,B 0,C 180,E1 809.997,E2 809.997} C_VEL
LIN {X 0,Y 609.864,Z 526.81,A -85,B 0,C 180,E1 814.268,E2 814.268} C_VEL
LIN {X 0,Y 609.933,Z 526.81,A -85,B 0,C 180,E1 818.562,E2 818.562} C_VEL
LIN {X 0,Y 610.059,Z 526.81,A -85,B 0,C 180,E1 822.903,E2 822.903} C_VEL
LIN {X 0,Y 609.783,Z 526.81,A -85,B 0,C 180,E1 828.828,E2 828.828} C_VEL
LIN {X 0,Y 609.72,Z 526.81,A -85,B 0,C 180,E1 833.407,E2 833.407} C_VEL
LIN {X 0,Y 609.773,Z 526.81,A -85,B 0,C 180,E1 838.145,E2 838.145} C_VEL
LIN {X 0,Y 609.927,Z 526.81,A -85,B 0,C 180,E1 843.097,E2 843.097} C_VEL
LIN {X 0,Y 609.596,Z 526.81,A -85,B 0,C 180,E1 849.647,E2 849.647} C_VEL
LIN {X 0,Y 609.704,Z 526.81,A -85,B 0,C 180,E1 855.944,E2 855.944} C_VEL
LIN {X 0,Y 609.54,Z 526.81,A -85,B 0,C 180,E1 860.351,E2 860.351} C_VEL
LIN {X 0,Y 609.619,Z 526.81,A -85,B 0,C 180,E1 865.16,E2 865.16} C_VEL
LIN {X 0,Y 609.767,Z 526.81,A -85,B 0,C 180,E1 870.343,E2 870.343} C_VEL
LIN {X 0,Y 609.963,Z 526.81,A -85,B 0,C 180,E1 875.037,E2 875.037} C_VEL
LIN {X 0,Y 609.847,Z 526.81,A -85,B 0,C 180,E1 881.167,E2 881.167} C_VEL
LIN {X 0,Y 609.41,Z 526.81,A -85,B 0,C 180,E1 885.671,E2 885.671} C_VEL
LIN {X 0,Y 609.939,Z 526.81,A -85,B 0,C 180,E1 889.989,E2 889.989} C_VEL
LIN {X 0,Y 609.944,Z 526.81,A -85,B 0,C 180,E1 894.598,E2 894.598} C_VEL
LIN {X 0,Y 605.685,Z 526.81,A -85,B 0,C 180,E1 896.195,E2 896.195} C_VEL
LIN {X 0,Y 601.879,Z 526.81,A -85,B 0,C 180,E1 897.812,E2 897.812} C_VEL
LIN {X 0,Y 602.014,Z 526.81,A -85,B 0,C 180,E1 902.879,E2 902.879} C_VEL
LIN {X 0,Y 601.97,Z 526.81,A -85,B 0,C 180,E1 908.675,E2 908.675} C_VEL
LIN {X 0,Y 602.046,Z 526.81,A -85,B 0,C 180,E1 913.076,E2 913.076} C_VEL
LIN {X 0,Y 602.035,Z 526.81,A -85,B 0,C 180,E1 917.56,E2 917.56} C_VEL
LIN {X 0,Y 601.715,Z 526.81,A -85,B 0,C 180,E1 923.735,E2 923.735} C_VEL
LIN {X 0,Y 601.78,Z 526.81,A -85,B 0,C 180,E1 928.551,E2 928.551} C_VEL
LIN {X 0,Y 601.904,Z 526.81,A -85,B 0,C 180,E1 933.897,E2 933.897} C_VEL
LIN {X 0,Y 601.691,Z 526.81,A -85,B 0,C 180,E1 938.975,E2 938.975} C_VEL
LIN {X 0,Y 601.548,Z 526.81,A -85,B 0,C 180,E1 943.126,E2 943.126} C_VEL
LIN {X 0,Y 601.601,Z 526.81,A -85,B 0,C 180,E1 949.134,E2 949.134} C_VEL
LIN {X 0,Y 601.706,Z 526.81,A -85,B 0,C 180,E1 954.642,E2 954.642} C_VEL
LIN {X 0,Y 601.772,Z 526.81,A -85,B 0,C 180,E1 959.792,E2 959.792} C_VEL
LIN {X 0,Y 602.054,Z 526.81,A -85,B 0,C 180,E1 964.852,E2 964.852} C_VEL
LIN {X 0,Y 602.064,Z 526.81,A -85,B 0,C 180,E1 968.687,E2 968.687} C_VEL
LIN {X 0,Y 603.115,Z 606.154,A -85,B 0,C 180,E1 969.81,E2 969.81} C_VEL
LIN {X 0,Y 602.923,Z 638.931,A -85,B 0,C 180,E1 970.81,E2 970.81} C_VEL
LIN {X 0,Y 602.769,Z 670.627,A -85,B 0,C 180,E1 972.366,E2 972.366} C_VEL
LIN {X 0,Y 602.569,Z 699.522,A -85,B 0,C 180,E1 974.426,E2 974.426} C_VEL
LIN {X 0,Y 602.4,Z 724.69,A -85,B 0,C 180,E1 976.93,E2 976.93} C_VEL
LIN {X 0,Y 602.349,Z 743.815,A -85,B 0,C 180,E1 979.549,E2 979.549} C_VEL
LIN {X 0,Y 602.276,Z 758.575,A -85,B 0,C 180,E1 982.419,E2 982.419} C_VEL
LIN {X 0,Y 602.243,Z 769.078,A -85,B 0,C 180,E1 985.678,E2 985.678} C_VEL
LIN {X 0,Y 602.193,Z 773.419,A -85,B 0,C 180,E1 988.563,E2 988.563} C_VEL
LIN {X 0,Y 602.151,Z 773.414,A -85,B 0,C 180,E1 991.444,E2 991.444} C_VEL
LIN {X 0,Y 602.197,Z 769.064,A -85,B 0,C 180,E1 994.329,E2 994.329} C_VEL
LIN {X 0,Y 602.262,Z 758.546,A -85,B 0,C 180,E1 997.588,E2 997.588} C_VEL
LIN {X 0,Y 602.324,Z 742.739,A -85,B 0,C 180,E1 1000.626,E2 1000.626} C_VEL
LIN {X 0,Y 602.446,Z 721.419,A -85,B 0,C 180,E1 1003.446,E2 1003.446} C_VEL
LIN {X 0,Y 602.6,Z 696.011,A -85,B 0,C 180,E1 1005.861,E2 1005.861} C_VEL
LIN {X 0,Y 602.762,Z 667.26,A -85,B 0,C 180,E1 1007.83,E2 1007.83} C_VEL
LIN {X 0,Y 602.929,Z 635.096,A -85,B 0,C 180,E1 1009.341,E2 1009.341} C_VEL
LIN {X 0,Y 603.063,Z 600.807,A -85,B 0,C 180,E1 1010.298,E2 1010.298} C_VEL
LIN {X 0,Y 602.136,Z 526.81,A -85,B 0,C 180,E1 1011.325,E2 1011.325} C_VEL
LIN {X 0,Y 602.012,Z 526.81,A -85,B 0,C 180,E1 1015.316,E2 1015.316} C_VEL
LIN {X 0,Y 601.667,Z 526.81,A -85,B 0,C 180,E1 1021.188,E2 1021.188} C_VEL
LIN {X 0,Y 601.723,Z 526.81,A -85,B 0,C 180,E1 1027.153,E2 1027.153} C_VEL
LIN {X 0,Y 601.778,Z 526.81,A -85,B 0,C 180,E1 1033.154,E2 1033.154} C_VEL
LIN {X 0,Y 601.579,Z 526.81,A -85,B 0,C 180,E1 1039.136,E2 1039.136} C_VEL
LIN {X 0,Y 601.497,Z 526.81,A -85,B 0,C 180,E1 1043.664,E2 1043.664} C_VEL
LIN {X 0,Y 601.814,Z 526.81,A -85,B 0,C 180,E1 1048.115,E2 1048.115} C_VEL
LIN {X 0,Y 601.656,Z 526.81,A -85,B 0,C 180,E1 1053.072,E2 1053.072} C_VEL
LIN {X 0,Y 601.661,Z 526.81,A -85,B 0,C 180,E1 1058.616,E2 1058.616} C_VEL
LIN {X 0,Y 601.94,Z 526.81,A -85,B 0,C 180,E1 1062.917,E2 1062.917} C_VEL
LIN {X 0,Y 602.022,Z 526.81,A -85,B 0,C 180,E1 1067.856,E2 1067.856} C_VEL
LIN {X 0,Y 602.536,Z 552.918,A -85,B 0,C 180,E1 1068.839,E2 1068.839} C_VEL
LIN {X 0,Y 602.446,Z 576.424,A -85,B 0,C 180,E1 1070.329,E2 1070.329} C_VEL
LIN {X 0,Y 602.326,Z 595.904,A -85,B 0,C 180,E1 1072.24,E2 1072.24} C_VEL
LIN {X 0,Y 602.283,Z 609.336,A -85,B 0,C 180,E1 1074.234,E2 1074.234} C_VEL
LIN {X 0,Y 602.243,Z 619.599,A -85,B 0,C 180,E1 1076.762,E2 1076.762} C_VEL
LIN {X 0,Y 602.248,Z 623.152,A -85,B 0,C 180,E1 1078.564,E2 1078.564} C_VEL
LIN {X 0,Y 602.255,Z 623.995,A -85,B 0,C 180,E1 1080.004,E2 1080.004} C_VEL
LIN {X 0,Y 602.23,Z 621.916,A -85,B 0,C 180,E1 1082.166,E2 1082.166} C_VEL
LIN {X 0,Y 602.281,Z 614.13,A -85,B 0,C 180,E1 1084.691,E2 1084.691} C_VEL
LIN {X 0,Y 602.315,Z 600.498,A -85,B 0,C 180,E1 1087.076,E2 1087.076} C_VEL
LIN {X 0,Y 602.388,Z 581.775,A -85,B 0,C 180,E1 1089.133,E2 1089.133} C_VEL
LIN {X 0,Y 602.502,Z 559.389,A -85,B 0,C 180,E1 1090.73,E2 1090.73} C_VEL
LIN {X 0,Y 602.575,Z 533.411,A -85,B 0,C 180,E1 1091.853,E2 1091.853} C_VEL
LIN {X 0,Y 602.181,Z 526.81,A -85,B 0,C 180,E1 1092.115,E2 1092.115} C_VEL
LIN {X 0,Y 601.995,Z 526.81,A -85,B 0,C 180,E1 1097.57,E2 1097.57} C_VEL
LIN {X 0,Y 601.765,Z 526.81,A -85,B 0,C 180,E1 1103.742,E2 1103.742} C_VEL
LIN {X 0,Y 601.779,Z 526.81,A -85,B 0,C 180,E1 1108.561,E2 1108.561} C_VEL
LIN {X 0,Y 601.818,Z 526.81,A -85,B 0,C 180,E1 1113.872,E2 1113.872} C_VEL
LIN {X 0,Y 601.77,Z 526.81,A -85,B 0,C 180,E1 1118.98,E2 1118.98} C_VEL
LIN {X 0,Y 601.731,Z 526.81,A -85,B 0,C 180,E1 1125.203,E2 1125.203} C_VEL
LIN {X 0,Y 601.693,Z 526.81,A -85,B 0,C 180,E1 1131.013,E2 1131.013} C_VEL
LIN {X 0,Y 601.568,Z 526.81,A -85,B 0,C 180,E1 1136.161,E2 1136.161} C_VEL
LIN {X 0,Y 601.679,Z 526.81,A -85,B 0,C 180,E1 1141.434,E2 1141.434} C_VEL
LIN {X 0,Y 601.719,Z 526.81,A -85,B 0,C 180,E1 1146.256,E2 1146.256} C_VEL
LIN {X 0,Y 601.935,Z 526.81,A -85,B 0,C 180,E1 1150.91,E2 1150.91} C_VEL
LIN {X 0,Y 601.538,Z 526.81,A -85,B 0,C 180,E1 1155.418,E2 1155.418} C_VEL
LIN {X 0,Y 601.993,Z 526.81,A -85,B 0,C 180,E1 1159.856,E2 1159.856} C_VEL
LIN {X 0,Y 602.177,Z 526.81,A -85,B 0,C 180,E1 1164.224,E2 1164.224} C_VEL
LIN {X 0,Y 601.884,Z 526.81,A -85,B 0,C 180,E1 1169.997,E2 1169.997} C_VEL
LIN {X 0,Y 601.976,Z 526.81,A -85,B 0,C 180,E1 1174.324,E2 1174.324} C_VEL
LIN {X 0,Y 601.992,Z 526.81,A -85,B 0,C 180,E1 1178.676,E2 1178.676} C_VEL
LIN {X 0,Y 602.083,Z 526.81,A -85,B 0,C 180,E1 1183.077,E2 1183.077} C_VEL
LIN {X 0,Y 601.841,Z 526.81,A -85,B 0,C 180,E1 1189.086,E2 1189.086} C_VEL
LIN {X 0,Y 601.743,Z 526.81,A -85,B 0,C 180,E1 1193.736,E2 1193.736} C_VEL
LIN {X 0,Y 601.767,Z 526.81,A -85,B 0,C 180,E1 1198.554,E2 1198.554} C_VEL
LIN {X 0,Y 601.822,Z 526.81,A -85,B 0,C 180,E1 1203.876,E2 1203.876} C_VEL
LIN {X 0,Y 601.758,Z 526.81,A -85,B 0,C 180,E1 1208.973,E2 1208.973} C_VEL
LIN {X 0,Y 601.702,Z 526.81,A -85,B 0,C 180,E1 1215.202,E2 1215.202} C_VEL
LIN {X 0,Y 601.68,Z 526.81,A -85,B 0,C 180,E1 1221.013,E2 1221.013} C_VEL
LIN {X 0,Y 601.563,Z 526.81,A -85,B 0,C 180,E1 1226.152,E2 1226.152} C_VEL
LIN {X 0,Y 601.65,Z 526.81,A -85,B 0,C 180,E1 1231.433,E2 1231.433} C_VEL
LIN {X 0,Y 601.71,Z 526.81,A -85,B 0,C 180,E1 1236.255,E2 1236.255} C_VEL
LIN {X 0,Y 601.972,Z 526.81,A -85,B 0,C 180,E1 1240.911,E2 1240.911} C_VEL
LIN {X 0,Y 601.544,Z 526.81,A -85,B 0,C 180,E1 1245.418,E2 1245.418} C_VEL
LIN {X 0,Y 601.996,Z 526.81,A -85,B 0,C 180,E1 1249.856,E2 1249.856} C_VEL
LIN {X 0,Y 602.024,Z 526.81,A -85,B 0,C 180,E1 1254.576,E2 1254.576} C_VEL
LIN {X 0,Y 601.879,Z 526.81,A -85,B 0,C 180,E1 1257.812,E2 1257.812} C_VEL
LIN {X 0,Y 599.44,Z 526.81,A -85,B 0,C 180,E1 1259.042,E2 1259.042} C_VEL
LIN {X 0,Y 593.935,Z 526.81,A -85,B 0,C 180,E1 1260.88,E2 1260.88} C_VEL
LIN {X 0,Y 593.835,Z 526.81,A -85,B 0,C 180,E1 1261.093,E2 1261.093} C_VEL
LIN {X 0,Y 593.837,Z 526.81,A -85,B 0,C 180,E1 1265.849,E2 1265.849} C_VEL
LIN {X 0,Y 593.785,Z 526.81,A -85,B 0,C 180,E1 1270.277,E2 1270.277} C_VEL
LIN {X 0,Y 593.764,Z 526.81,A -85,B 0,C 180,E1 1274.768,E2 1274.768} C_VEL
LIN {X 0,Y 593.869,Z 526.81,A -85,B 0,C 180,E1 1279.395,E2 1279.395} C_VEL
LIN {X 0,Y 593.791,Z 526.81,A -85,B 0,C 180,E1 1284.071,E2 1284.071} C_VEL
LIN {X 0,Y 593.782,Z 526.81,A -85,B 0,C 180,E1 1288.971,E2 1288.971} C_VEL
LIN {X 0,Y 593.98,Z 526.81,A -85,B 0,C 180,E1 1294.103,E2 1294.103} C_VEL
LIN {X 0,Y 593.712,Z 526.81,A -85,B 0,C 180,E1 1300.094,E2 1300.094} C_VEL
LIN {X 0,Y 593.515,Z 526.81,A -85,B 0,C 180,E1 1305.575,E2 1305.575} C_VEL
LIN {X 0,Y 593.532,Z 526.81,A -85,B 0,C 180,E1 1310.381,E2 1310.381} C_VEL
LIN {X 0,Y 593.641,Z 526.81,A -85,B 0,C 180,E1 1315.872,E2 1315.872} C_VEL
LIN {X 0,Y 593.735,Z 526.81,A -85,B 0,C 180,E1 1321.023,E2 1321.023} C_VEL
LIN {X 0,Y 593.95,Z 526.81,A -85,B 0,C 180,E1 1325.933,E2 1325.933} C_VEL
LIN {X 0,Y 594.105,Z 526.81,A -85,B 0,C 180,E1 1328.376,E2 1328.376} C_VEL
LIN {X 0,Y 595.534,Z 537.872,A -85,B 0,C 180,E1 1328.585,E2 1328.585} C_VEL
LIN {X 0,Y 595.68,Z 606.98,A -85,B 0,C 180,E1 1329.566,E2 1329.566} C_VEL
LIN {X 0,Y 595.428,Z 641.324,A -85,B 0,C 180,E1 1330.655,E2 1330.655} C_VEL
LIN {X 0,Y 595.085,Z 673.602,A -85,B 0,C 180,E1 1332.318,E2 1332.318} C_VEL
LIN {X 0,Y 594.769,Z 702.741,A -85,B 0,C 180,E1 1334.5,E2 1334.5} C_VEL
LIN {X 0,Y 594.548,Z 727.777,A -85,B 0,C 180,E1 1337.128,E2 1337.128} C_VEL
LIN {X 0,Y 594.404,Z 747.897,A -85,B 0,C 180,E1 1340.103,E2 1340.103} C_VEL
LIN {X 0,Y 594.332,Z 761.898,A -85,B 0,C 180,E1 1343.175,E2 1343.175} C_VEL
LIN {X 0,Y 594.268,Z 770.615,A -85,B 0,C 180,E1 1346.352,E2 1346.352} C_VEL
LIN {X 0,Y 594.289,Z 773.419,A -85,B 0,C 180,E1 1348.544,E2 1348.544} C_VEL
LIN {X 0,Y 594.248,Z 773.414,A -85,B 0,C 180,E1 1351.463,E2 1351.463} C_VEL
LIN {X 0,Y 594.299,Z 769.065,A -85,B 0,C 180,E1 1354.387,E2 1354.387} C_VEL
LIN {X 0,Y 594.395,Z 758.546,A -85,B 0,C 180,E1 1357.689,E2 1357.689} C_VEL
LIN {X 0,Y 594.472,Z 742.197,A -85,B 0,C 180,E1 1360.852,E2 1360.852} C_VEL
LIN {X 0,Y 594.64,Z 721.542,A -85,B 0,C 180,E1 1363.612,E2 1363.612} C_VEL
LIN {X 0,Y 594.902,Z 696.014,A -85,B 0,C 180,E1 1366.071,E2 1366.071} C_VEL
LIN {X 0,Y 595.199,Z 667.264,A -85,B 0,C 180,E1 1368.064,E2 1368.064} C_VEL
LIN {X 0,Y 595.426,Z 635.457,A -85,B 0,C 180,E1 1369.58,E2 1369.58} C_VEL
LIN {X 0,Y 595.67,Z 601.277,A -85,B 0,C 180,E1 1370.551,E2 1370.551} C_VEL
LIN {X 0,Y 594.842,Z 529.939,A -85,B 0,C 180,E1 1371.542,E2 1371.542} C_VEL
LIN {X 0,Y 594.136,Z 526.81,A -85,B 0,C 180,E1 1371.638,E2 1371.638} C_VEL
LIN {X 0,Y 593.707,Z 526.81,A -85,B 0,C 180,E1 1377.329,E2 1377.329} C_VEL
LIN {X 0,Y 593.594,Z 526.81,A -85,B 0,C 180,E1 1382.392,E2 1382.392} C_VEL
LIN {X 0,Y 593.775,Z 526.81,A -85,B 0,C 180,E1 1387.782,E2 1387.782} C_VEL
LIN {X 0,Y 593.832,Z 526.81,A -85,B 0,C 180,E1 1393.509,E2 1393.509} C_VEL
LIN {X 0,Y 593.635,Z 526.81,A -85,B 0,C 180,E1 1398.47,E2 1398.47} C_VEL
LIN {X 0,Y 593.637,Z 526.81,A -85,B 0,C 180,E1 1404.091,E2 1404.091} C_VEL
LIN {X 0,Y 593.826,Z 526.81,A -85,B 0,C 180,E1 1409.347,E2 1409.347} C_VEL
LIN {X 0,Y 593.704,Z 526.81,A -85,B 0,C 180,E1 1414.314,E2 1414.314} C_VEL
LIN {X 0,Y 593.729,Z 526.81,A -85,B 0,C 180,E1 1419.089,E2 1419.089} C_VEL
LIN {X 0,Y 593.804,Z 526.81,A -85,B 0,C 180,E1 1423.717,E2 1423.717} C_VEL
LIN {X 0,Y 594.16,Z 526.81,A -85,B 0,C 180,E1 1427.683,E2 1427.683} C_VEL
LIN {X 0,Y 594.768,Z 553.395,A -85,B 0,C 180,E1 1428.716,E2 1428.716} C_VEL
LIN {X 0,Y 594.63,Z 576.418,A -85,B 0,C 180,E1 1430.201,E2 1430.201} C_VEL
LIN {X 0,Y 594.476,Z 595.9,A -85,B 0,C 180,E1 1432.137,E2 1432.137} C_VEL
LIN {X 0,Y 594.397,Z 609.334,A -85,B 0,C 180,E1 1434.157,E2 1434.157} C_VEL
LIN {X 0,Y 594.35,Z 619.597,A -85,B 0,C 180,E1 1436.719,E2 1436.719} C_VEL
LIN {X 0,Y 594.348,Z 623.152,A -85,B 0,C 180,E1 1438.545,E2 1438.545} C_VEL
LIN {X 0,Y 594.356,Z 623.996,A -85,B 0,C 180,E1 1440.004,E2 1440.004} C_VEL
LIN {X 0,Y 594.33,Z 621.917,A -85,B 0,C 180,E1 1442.194,E2 1442.194} C_VEL
LIN {X 0,Y 594.411,Z 614.133,A -85,B 0,C 180,E1 1444.753,E2 1444.753} C_VEL
LIN {X 0,Y 594.442,Z 601.148,A -85,B 0,C 180,E1 1447.081,E2 1447.081} C_VEL
LIN {X 0,Y 594.557,Z 582.826,A -85,B 0,C 180,E1 1449.162,E2 1449.162} C_VEL
LIN {X 0,Y 594.721,Z 559.733,A -85,B 0,C 180,E1 1450.853,E2 1450.853} C_VEL
LIN {X 0,Y 594.859,Z 534.144,A -85,B 0,C 180,E1 1451.986,E2 1451.986} C_VEL
LIN {X 0,Y 594.232,Z 526.81,A -85,B 0,C 180,E1 1452.232,E2 1452.232} C_VEL
LIN {X 0,Y 594.044,Z 526.81,A -85,B 0,C 180,E1 1457.813,E2 1457.813} C_VEL
LIN {X 0,Y 593.858,Z 526.81,A -85,B 0,C 180,E1 1463.38,E2 1463.38} C_VEL
LIN {X 0,Y 593.769,Z 526.81,A -85,B 0,C 180,E1 1468.982,E2 1468.982} C_VEL
LIN {X 0,Y 593.876,Z 526.81,A -85,B 0,C 180,E1 1474.12,E2 1474.12} C_VEL
LIN {X 0,Y 593.683,Z 526.81,A -85,B 0,C 180,E1 1480.08,E2 1480.08} C_VEL
LIN {X 0,Y 593.799,Z 526.81,A -85,B 0,C 180,E1 1485.56,E2 1485.56} C_VEL
LIN {X 0,Y 593.734,Z 526.81,A -85,B 0,C 180,E1 1490.388,E2 1490.388} C_VEL
LIN {X 0,Y 593.678,Z 526.81,A -85,B 0,C 180,E1 1495.866,E2 1495.866} C_VEL
LIN {X 0,Y 593.769,Z 526.81,A -85,B 0,C 180,E1 1501.017,E2 1501.017} C_VEL
LIN {X 0,Y 593.893,Z 526.81,A -85,B 0,C 180,E1 1505.923,E2 1505.923} C_VEL
LIN {X 0,Y 594.033,Z 526.81,A -85,B 0,C 180,E1 1510.646,E2 1510.646} C_VEL
LIN {X 0,Y 593.698,Z 526.81,A -85,B 0,C 180,E1 1515.221,E2 1515.221} C_VEL
LIN {X 0,Y 594.054,Z 526.81,A -85,B 0,C 180,E1 1519.719,E2 1519.719} C_VEL
LIN {X 0,Y 594.24,Z 526.81,A -85,B 0,C 180,E1 1524.147,E2 1524.147} C_VEL
LIN {X 0,Y 593.984,Z 526.81,A -85,B 0,C 180,E1 1529.997,E2 1529.997} C_VEL
LIN {X 0,Y 594.059,Z 526.81,A -85,B 0,C 180,E1 1534.382,E2 1534.382} C_VEL
LIN {X 0,Y 594.074,Z 526.81,A -85,B 0,C 180,E1 1538.793,E2 1538.793} C_VEL
LIN {X 0,Y 593.877,Z 526.81,A -85,B 0,C 180,E1 1544.344,E2 1544.344} C_VEL
LIN {X 0,Y 593.909,Z 526.81,A -85,B 0,C 180,E1 1549.39,E2 1549.39} C_VEL
LIN {X 0,Y 593.821,Z 526.81,A -85,B 0,C 180,E1 1554.072,E2 1554.072} C_VEL
LIN {X 0,Y 593.757,Z 526.81,A -85,B 0,C 180,E1 1558.975,E2 1558.975} C_VEL
LIN {X 0,Y 593.881,Z 526.81,A -85,B 0,C 180,E1 1564.112,E2 1564.112} C_VEL
LIN {X 0,Y 593.661,Z 526.81,A -85,B 0,C 180,E1 1570.079,E2 1570.079} C_VEL
LIN {X 0,Y 593.767,Z 526.81,A -85,B 0,C 180,E1 1575.555,E2 1575.555} C_VEL
LIN {X 0,Y 593.721,Z 526.81,A -85,B 0,C 180,E1 1580.388,E2 1580.388} C_VEL
LIN {X 0,Y 593.675,Z 526.81,A -85,B 0,C 180,E1 1585.867,E2 1585.867} C_VEL
LIN {X 0,Y 593.744,Z 526.81,A -85,B 0,C 180,E1 1591.016,E2 1591.016} C_VEL
LIN {X 0,Y 593.876,Z 526.81,A -85,B 0,C 180,E1 1595.922,E2 1595.922} C_VEL
LIN {X 0,Y 594.039,Z 526.81,A -85,B 0,C 180,E1 1600.646,E2 1600.646} C_VEL
LIN {X 0,Y 593.694,Z 526.81,A -85,B 0,C 180,E1 1605.221,E2 1605.221} C_VEL
LIN {X 0,Y 594.061,Z 526.81,A -85,B 0,C 180,E1 1609.719,E2 1609.719} C_VEL
LIN {X 0,Y 594.214,Z 526.81,A -85,B 0,C 180,E1 1614.146,E2 1614.146} C_VEL
LIN {X 0,Y 593.965,Z 526.81,A -85,B 0,C 180,E1 1619.995,E2 1619.995} C_VEL
LIN {X 0,Y 593.835,Z 526.81,A -85,B 0,C 180,E1 1621.093,E2 1621.093} C_VEL
LIN {X 0,Y 589.953,Z 526.81,A -85,B 0,C 180,E1 1622.747,E2 1622.747} C_VEL
LIN {X 0,Y 586.15,Z 526.81,A -85,B 0,C 180,E1 1624.424,E2 1624.424} C_VEL
LIN {X 0,Y 586.11,Z 526.81,A -85,B 0,C 180,E1 1628.911,E2 1628.911} C_VEL
LIN {X 0,Y 586.132,Z 526.81,A -85,B 0,C 180,E1 1633.438,E2 1633.438} C_VEL
LIN {X 0,Y 586.117,Z 526.81,A -85,B 0,C 180,E1 1638.053,E2 1638.053} C_VEL
LIN {X 0,Y 585.963,Z 526.81,A -85,B 0,C 180,E1 1642.798,E2 1642.798} C_VEL
LIN {X 0,Y 585.863,Z 526.81,A -85,B 0,C 180,E1 1648.525,E2 1648.525} C_VEL
LIN {X 0,Y 586.022,Z 526.81,A -85,B 0,C 180,E1 1654.631,E2 1654.631} C_VEL
LIN {X 0,Y 585.823,Z 526.81,A -85,B 0,C 180,E1 1660.242,E2 1660.242} C_VEL
LIN {X 0,Y 585.709,Z 526.81,A -85,B 0,C 180,E1 1666.36,E2 1666.36} C_VEL
LIN {X 0,Y 585.655,Z 526.81,A -85,B 0,C 180,E1 1671.655,E2 1671.655} C_VEL
LIN {X 0,Y 585.706,Z 526.81,A -85,B 0,C 180,E1 1677.126,E2 1677.126} C_VEL
LIN {X 0,Y 585.772,Z 526.81,A -85,B 0,C 180,E1 1682.277,E2 1682.277} C_VEL
LIN {X 0,Y 586.009,Z 526.81,A -85,B 0,C 180,E1 1687.201,E2 1687.201} C_VEL
LIN {X 0,Y 586.129,Z 527.026,A -85,B 0,C 180,E1 1688.084,E2 1688.084} C_VEL
LIN {X 0,Y 588.177,Z 537.882,A -85,B 0,C 180,E1 1688.304,E2 1688.304} C_VEL
LIN {X 0,Y 588.261,Z 607.797,A -85,B 0,C 180,E1 1689.317,E2 1689.317} C_VEL
LIN {X 0,Y 587.933,Z 641.326,A -85,B 0,C 180,E1 1690.398,E2 1690.398} C_VEL
LIN {X 0,Y 587.524,Z 673.425,A -85,B 0,C 180,E1 1692.071,E2 1692.071} C_VEL
LIN {X 0,Y 587.105,Z 702.742,A -85,B 0,C 180,E1 1694.293,E2 1694.293} C_VEL
LIN {X 0,Y 586.745,Z 727.779,A -85,B 0,C 180,E1 1696.954,E2 1696.954} C_VEL
LIN {X 0,Y 586.55,Z 747.897,A -85,B 0,C 180,E1 1699.969,E2 1699.969} C_VEL
LIN {X 0,Y 586.456,Z 761.497,A -85,B 0,C 180,E1 1702.971,E2 1702.971} C_VEL
LIN {X 0,Y 586.385,Z 770.615,A -85,B 0,C 180,E1 1706.302,E2 1706.302} C_VEL
LIN {X 0,Y 586.385,Z 773.419,A -85,B 0,C 180,E1 1708.524,E2 1708.524} C_VEL
LIN {X 0,Y 586.348,Z 773.415,A -85,B 0,C 180,E1 1711.483,E2 1711.483} C_VEL
LIN {X 0,Y 586.403,Z 769.064,A -85,B 0,C 180,E1 1714.446,E2 1714.446} C_VEL
LIN {X 0,Y 586.507,Z 758.545,A -85,B 0,C 180,E1 1717.793,E2 1717.793} C_VEL
LIN {X 0,Y 586.614,Z 743.045,A -85,B 0,C 180,E1 1720.866,E2 1720.866} C_VEL
LIN {X 0,Y 586.858,Z 721.867,A -85,B 0,C 180,E1 1723.757,E2 1723.757} C_VEL
LIN {X 0,Y 587.226,Z 696.016,A -85,B 0,C 180,E1 1726.287,E2 1726.287} C_VEL
LIN {X 0,Y 587.614,Z 667.267,A -85,B 0,C 180,E1 1728.306,E2 1728.306} C_VEL
LIN {X 0,Y 587.942,Z 635.455,A -85,B 0,C 180,E1 1729.84,E2 1729.84} C_VEL
LIN {X 0,Y 588.251,Z 600.341,A -85,B 0,C 180,E1 1730.841,E2 1730.841} C_VEL
LIN {X 0,Y 587.485,Z 531.695,A -85,B 0,C 180,E1 1731.803,E2 1731.803} C_VEL
LIN {X 0,Y 586.165,Z 526.81,A -85,B 0,C 180,E1 1731.967,E2 1731.967} C_VEL
LIN {X 0,Y 586.002,Z 526.81,A -85,B 0,C 180,E1 1736.059,E2 1736.059} C_VEL
LIN {X 0,Y 585.767,Z 526.81,A -85,B 0,C 180,E1 1741.477,E2 1741.477} C_VEL
LIN {X 0,Y 585.849,Z 526.81,A -85,B 0,C 180,E1 1746.77,E2 1746.77} C_VEL
LIN {X 0,Y 585.912,Z 526.81,A -85,B 0,C 180,E1 1752.216,E2 1752.216} C_VEL
LIN {X 0,Y 585.746,Z 526.81,A -85,B 0,C 180,E1 1757.782,E2 1757.782} C_VEL
LIN {X 0,Y 585.714,Z 526.81,A -85,B 0,C 180,E1 1763.265,E2 1763.265} C_VEL
LIN {X 0,Y 585.902,Z 526.81,A -85,B 0,C 180,E1 1768.521,E2 1768.521} C_VEL
LIN {X 0,Y 585.81,Z 526.81,A -85,B 0,C 180,E1 1773.942,E2 1773.942} C_VEL
LIN {X 0,Y 585.805,Z 526.81,A -85,B 0,C 180,E1 1778.793,E2 1778.793} C_VEL
LIN {X 0,Y 585.915,Z 526.81,A -85,B 0,C 180,E1 1783.492,E2 1783.492} C_VEL
LIN {X 0,Y 586.202,Z 526.81,A -85,B 0,C 180,E1 1787.513,E2 1787.513} C_VEL
LIN {X 0,Y 587.041,Z 552.731,A -85,B 0,C 180,E1 1788.532,E2 1788.532} C_VEL
LIN {X 0,Y 586.815,Z 576.412,A -85,B 0,C 180,E1 1790.069,E2 1790.069} C_VEL
LIN {X 0,Y 586.61,Z 595.895,A -85,B 0,C 180,E1 1792.031,E2 1792.031} C_VEL
LIN {X 0,Y 586.531,Z 609.331,A -85,B 0,C 180,E1 1794.078,E2 1794.078} C_VEL
LIN {X 0,Y 586.458,Z 619.595,A -85,B 0,C 180,E1 1796.675,E2 1796.675} C_VEL
LIN {X 0,Y 586.451,Z 623.152,A -85,B 0,C 180,E1 1798.525,E2 1798.525} C_VEL
LIN {X 0,Y 586.456,Z 623.996,A -85,B 0,C 180,E1 1800.005,E2 1800.005} C_VEL
LIN {X 0,Y 586.439,Z 621.918,A -85,B 0,C 180,E1 1802.224,E2 1802.224} C_VEL
LIN {X 0,Y 586.52,Z 614.135,A -85,B 0,C 180,E1 1804.817,E2 1804.817} C_VEL
LIN {X 0,Y 586.58,Z 600.723,A -85,B 0,C 180,E1 1807.237,E2 1807.237} C_VEL
LIN {X 0,Y 586.739,Z 582.833,A -85,B 0,C 180,E1 1809.285,E2 1809.285} C_VEL
LIN {X 0,Y 586.933,Z 559.917,A -85,B 0,C 180,E1 1810.989,E2 1810.989} C_VEL
LIN {X 0,Y 587.119,Z 534.077,A -85,B 0,C 180,E1 1812.149,E2 1812.149} C_VEL
LIN {X 0,Y 586.254,Z 526.81,A -85,B 0,C 180,E1 1812.407,E2 1812.407} C_VEL
LIN {X 0,Y 586.098,Z 526.81,A -85,B 0,C 180,E1 1818.063,E2 1818.063} C_VEL
LIN {X 0,Y 586.011,Z 526.81,A -85,B 0,C 180,E1 1822.806,E2 1822.806} C_VEL
LIN {X 0,Y 585.845,Z 526.81,A -85,B 0,C 180,E1 1828.507,E2 1828.507} C_VEL
LIN {X 0,Y 585.872,Z 526.81,A -85,B 0,C 180,E1 1834.652,E2 1834.652} C_VEL
LIN {X 0,Y 585.769,Z 526.81,A -85,B 0,C 180,E1 1840.258,E2 1840.258} C_VEL
LIN {X 0,Y 585.935,Z 526.81,A -85,B 0,C 180,E1 1846.35,E2 1846.35} C_VEL
LIN {X 0,Y 585.851,Z 526.81,A -85,B 0,C 180,E1 1851.661,E2 1851.661} C_VEL
LIN {X 0,Y 585.748,Z 526.81,A -85,B 0,C 180,E1 1857.12,E2 1857.12} C_VEL
LIN {X 0,Y 585.805,Z 526.81,A -85,B 0,C 180,E1 1862.271,E2 1862.271} C_VEL
LIN {X 0,Y 585.847,Z 526.81,A -85,B 0,C 180,E1 1867.187,E2 1867.187} C_VEL
LIN {X 0,Y 586.091,Z 526.81,A -85,B 0,C 180,E1 1871.937,E2 1871.937} C_VEL
LIN {X 0,Y 585.819,Z 526.81,A -85,B 0,C 180,E1 1878.064,E2 1878.064} C_VEL
LIN {X 0,Y 586.315,Z 526.81,A -85,B 0,C 180,E1 1884.068,E2 1884.068} C_VEL
LIN {X 0,Y 586.094,Z 526.81,A -85,B 0,C 180,E1 1889.996,E2 1889.996} C_VEL
LIN {X 0,Y 586.149,Z 526.81,A -85,B 0,C 180,E1 1894.441,E2 1894.441} C_VEL
LIN {X 0,Y 586.137,Z 526.81,A -85,B 0,C 180,E1 1898.913,E2 1898.913} C_VEL
LIN {X 0,Y 586.174,Z 526.81,A -85,B 0,C 180,E1 1903.439,E2 1903.439} C_VEL
LIN {X 0,Y 585.998,Z 526.81,A -85,B 0,C 180,E1 1909.623,E2 1909.623} C_VEL
LIN {X 0,Y 585.858,Z 526.81,A -85,B 0,C 180,E1 1914.421,E2 1914.421} C_VEL
LIN {X 0,Y 585.781,Z 526.81,A -85,B 0,C 180,E1 1919.408,E2 1919.408} C_VEL
LIN {X 0,Y 585.872,Z 526.81,A -85,B 0,C 180,E1 1924.645,E2 1924.645} C_VEL
LIN {X 0,Y 585.745,Z 526.81,A -85,B 0,C 180,E1 1930.252,E2 1930.252} C_VEL
LIN {X 0,Y 585.892,Z 526.81,A -85,B 0,C 180,E1 1936.346,E2 1936.346} C_VEL
LIN {X 0,Y 585.812,Z 526.81,A -85,B 0,C 180,E1 1941.659,E2 1941.659} C_VEL
LIN {X 0,Y 585.747,Z 526.81,A -85,B 0,C 180,E1 1947.121,E2 1947.121} C_VEL
LIN {X 0,Y 585.769,Z 526.81,A -85,B 0,C 180,E1 1952.27,E2 1952.27} C_VEL
LIN {X 0,Y 585.85,Z 526.81,A -85,B 0,C 180,E1 1957.187,E2 1957.187} C_VEL
LIN {X 0,Y 586.128,Z 526.81,A -85,B 0,C 180,E1 1961.938,E2 1961.938} C_VEL
LIN {X 0,Y 585.833,Z 526.81,A -85,B 0,C 180,E1 1968.064,E2 1968.064} C_VEL
LIN {X 0,Y 586.289,Z 526.81,A -85,B 0,C 180,E1 1974.067,E2 1974.067} C_VEL
LIN {X 0,Y 586.074,Z 526.81,A -85,B 0,C 180,E1 1979.995,E2 1979.995} C_VEL
LIN {X 0,Y 586.15,Z 526.81,A -85,B 0,C 180,E1 1984.424,E2 1984.424} C_VEL
LIN {X 0,Y 583.672,Z 526.81,A -85,B 0,C 180,E1 1985.68,E2 1985.68} C_VEL
LIN {X 0,Y 578.246,Z 526.81,A -85,B 0,C 180,E1 1987.56,E2 1987.56} C_VEL
LIN {X 0,Y 578.137,Z 526.81,A -85,B 0,C 180,E1 1987.778,E2 1987.778} C_VEL
LIN {X 0,Y 578.173,Z 526.81,A -85,B 0,C 180,E1 1993.626,E2 1993.626} C_VEL
LIN {X 0,Y 578.069,Z 526.81,A -85,B 0,C 180,E1 1999.466,E2 1999.466} C_VEL
LIN {X 0,Y 577.928,Z 526.81,A -85,B 0,C 180,E1 2004.776,E2 2004.776} C_VEL
LIN {X 0,Y 577.857,Z 526.81,A -85,B 0,C 180,E1 2010.165,E2 2010.165} C_VEL
LIN {X 0,Y 578.01,Z 526.81,A -85,B 0,C 180,E1 2015.181,E2 2015.181} C_VEL
LIN {X 0,Y 577.882,Z 526.81,A -85,B 0,C 180,E1 2020.911,E2 2020.911} C_VEL
LIN {X 0,Y 577.825,Z 526.81,A -85,B 0,C 180,E1 2027.186,E2 2027.186} C_VEL
LIN {X 0,Y 577.837,Z 526.81,A -85,B 0,C 180,E1 2032.944,E2 2032.944} C_VEL
LIN {X 0,Y 577.872,Z 526.81,A -85,B 0,C 180,E1 2038.402,E2 2038.402} C_VEL
LIN {X 0,Y 577.994,Z 526.81,A -85,B 0,C 180,E1 2043.56,E2 2043.56} C_VEL
LIN {X 0,Y 578.227,Z 527.56,A -85,B 0,C 180,E1 2047.776,E2 2047.776} C_VEL
LIN {X 0,Y 580.811,Z 536.151,A -85,B 0,C 180,E1 2047.992,E2 2047.992} C_VEL
LIN {X 0,Y 580.86,Z 608.303,A -85,B 0,C 180,E1 2049.054,E2 2049.054} C_VEL
LIN {X 0,Y 580.458,Z 642.479,A -85,B 0,C 180,E1 2050.182,E2 2050.182} C_VEL
LIN {X 0,Y 579.922,Z 673.996,A -85,B 0,C 180,E1 2051.864,E2 2051.864} C_VEL
LIN {X 0,Y 579.4,Z 702.74,A -85,B 0,C 180,E1 2054.078,E2 2054.078} C_VEL
LIN {X 0,Y 578.952,Z 727.78,A -85,B 0,C 180,E1 2056.776,E2 2056.776} C_VEL
LIN {X 0,Y 578.7,Z 747.897,A -85,B 0,C 180,E1 2059.832,E2 2059.832} C_VEL
LIN {X 0,Y 578.571,Z 761.588,A -85,B 0,C 180,E1 2062.901,E2 2062.901} C_VEL
LIN {X 0,Y 578.508,Z 770.615,A -85,B 0,C 180,E1 2066.252,E2 2066.252} C_VEL
LIN {X 0,Y 578.482,Z 773.42,A -85,B 0,C 180,E1 2068.504,E2 2068.504} C_VEL
LIN {X 0,Y 578.445,Z 773.415,A -85,B 0,C 180,E1 2071.503,E2 2071.503} C_VEL
LIN {X 0,Y 578.508,Z 769.064,A -85,B 0,C 180,E1 2074.507,E2 2074.507} C_VEL
LIN {X 0,Y 578.622,Z 758.545,A -85,B 0,C 180,E1 2077.9,E2 2077.9} C_VEL
LIN {X 0,Y 578.791,Z 742.432,A -85,B 0,C 180,E1 2081.112,E2 2081.112} C_VEL
LIN {X 0,Y 579.114,Z 721.095,A -85,B 0,C 180,E1 2084.038,E2 2084.038} C_VEL
LIN {X 0,Y 579.576,Z 694.865,A -85,B 0,C 180,E1 2086.606,E2 2086.606} C_VEL
LIN {X 0,Y 580.047,Z 665.585,A -85,B 0,C 180,E1 2088.652,E2 2088.652} C_VEL
LIN {X 0,Y 580.577,Z 633.391,A -85,B 0,C 180,E1 2090.183,E2 2090.183} C_VEL
LIN {X 0,Y 580.873,Z 598.61,A -85,B 0,C 180,E1 2091.154,E2 2091.154} C_VEL
LIN {X 0,Y 580.11,Z 533.296,A -85,B 0,C 180,E1 2092.073,E2 2092.073} C_VEL
LIN {X 0,Y 578.211,Z 526.81,A -85,B 0,C 180,E1 2092.304,E2 2092.304} C_VEL
LIN {X 0,Y 577.92,Z 526.81,A -85,B 0,C 180,E1 2097.048,E2 2097.048} C_VEL
LIN {X 0,Y 577.804,Z 526.81,A -85,B 0,C 180,E1 2103.029,E2 2103.029} C_VEL
LIN {X 0,Y 577.898,Z 526.81,A -85,B 0,C 180,E1 2108.965,E2 2108.965} C_VEL
LIN {X 0,Y 577.95,Z 526.81,A -85,B 0,C 180,E1 2115.023,E2 2115.023} C_VEL
LIN {X 0,Y 577.882,Z 526.81,A -85,B 0,C 180,E1 2121.046,E2 2121.046} C_VEL
LIN {X 0,Y 578.091,Z 526.81,A -85,B 0,C 180,E1 2126.947,E2 2126.947} C_VEL
LIN {X 0,Y 577.883,Z 526.81,A -85,B 0,C 180,E1 2132.983,E2 2132.983} C_VEL
LIN {X 0,Y 577.931,Z 526.81,A -85,B 0,C 180,E1 2138.489,E2 2138.489} C_VEL
LIN {X 0,Y 578.056,Z 526.81,A -85,B 0,C 180,E1 2143.26,E2 2143.26} C_VEL
LIN {X 0,Y 578.28,Z 526.81,A -85,B 0,C 180,E1 2147.339,E2 2147.339} C_VEL
LIN {X 0,Y 579.316,Z 549.924,A -85,B 0,C 180,E1 2148.237,E2 2148.237} C_VEL
LIN {X 0,Y 579.004,Z 574.082,A -85,B 0,C 180,E1 2149.744,E2 2149.744} C_VEL
LIN {X 0,Y 578.776,Z 594.376,A -85,B 0,C 180,E1 2151.733,E2 2151.733} C_VEL
LIN {X 0,Y 578.655,Z 609.328,A -85,B 0,C 180,E1 2153.997,E2 2153.997} C_VEL
LIN {X 0,Y 578.58,Z 619.593,A -85,B 0,C 180,E1 2156.629,E2 2156.629} C_VEL
LIN {X 0,Y 578.551,Z 623.152,A -85,B 0,C 180,E1 2158.505,E2 2158.505} C_VEL
LIN {X 0,Y 578.556,Z 623.996,A -85,B 0,C 180,E1 2160.005,E2 2160.005} C_VEL
LIN {X 0,Y 578.545,Z 621.919,A -85,B 0,C 180,E1 2162.254,E2 2162.254} C_VEL
LIN {X 0,Y 578.639,Z 614.138,A -85,B 0,C 180,E1 2164.883,E2 2164.883} C_VEL
LIN {X 0,Y 578.73,Z 600.756,A -85,B 0,C 180,E1 2167.332,E2 2167.332} C_VEL
LIN {X 0,Y 578.901,Z 582.84,A -85,B 0,C 180,E1 2169.412,E2 2169.412} C_VEL
LIN {X 0,Y 579.155,Z 559.508,A -85,B 0,C 180,E1 2171.163,E2 2171.163} C_VEL
LIN {X 0,Y 579.392,Z 534.18,A -85,B 0,C 180,E1 2172.31,E2 2172.31} C_VEL
LIN {X 0,Y 578.277,Z 526.81,A -85,B 0,C 180,E1 2172.575,E2 2172.575} C_VEL
LIN {X 0,Y 578.152,Z 526.81,A -85,B 0,C 180,E1 2178.32,E2 2178.32} C_VEL
LIN {X 0,Y 578.017,Z 526.81,A -85,B 0,C 180,E1 2183.529,E2 2183.529} C_VEL
LIN {X 0,Y 577.973,Z 526.81,A -85,B 0,C 180,E1 2188.137,E2 2188.137} C_VEL
LIN {X 0,Y 578.035,Z 526.81,A -85,B 0,C 180,E1 2193.375,E2 2193.375} C_VEL
LIN {X 0,Y 577.866,Z 526.81,A -85,B 0,C 180,E1 2198.967,E2 2198.967} C_VEL
LIN {X 0,Y 577.954,Z 526.81,A -85,B 0,C 180,E1 2205.021,E2 2205.021} C_VEL
LIN {X 0,Y 577.912,Z 526.81,A -85,B 0,C 180,E1 2211.036,E2 2211.036} C_VEL
LIN {X 0,Y 577.86,Z 526.81,A -85,B 0,C 180,E1 2216.98,E2 2216.98} C_VEL
LIN {X 0,Y 577.917,Z 526.81,A -85,B 0,C 180,E1 2221.859,E2 2221.859} C_VEL
LIN {X 0,Y 577.935,Z 526.81,A -85,B 0,C 180,E1 2226.857,E2 2226.857} C_VEL
LIN {X 0,Y 578.165,Z 526.81,A -85,B 0,C 180,E1 2231.681,E2 2231.681} C_VEL
LIN {X 0,Y 577.877,Z 526.81,A -85,B 0,C 180,E1 2237.897,E2 2237.897} C_VEL
LIN {X 0,Y 578.389,Z 526.81,A -85,B 0,C 180,E1 2243.986,E2 2243.986} C_VEL
LIN {X 0,Y 578.193,Z 526.81,A -85,B 0,C 180,E1 2249.996,E2 2249.996} C_VEL
LIN {X 0,Y 578.234,Z 526.81,A -85,B 0,C 180,E1 2254.502,E2 2254.502} C_VEL
LIN {X 0,Y 578.204,Z 526.81,A -85,B 0,C 180,E1 2259.036,E2 2259.036} C_VEL
LIN {X 0,Y 578.074,Z 526.81,A -85,B 0,C 180,E1 2264.276,E2 2264.276} C_VEL
LIN {X 0,Y 578.065,Z 526.81,A -85,B 0,C 180,E1 2269.903,E2 2269.903} C_VEL
LIN {X 0,Y 577.952,Z 526.81,A -85,B 0,C 180,E1 2274.777,E2 2274.777} C_VEL
LIN {X 0,Y 577.816,Z 526.81,A -85,B 0,C 180,E1 2280.146,E2 2280.146} C_VEL
LIN {X 0,Y 577.851,Z 526.81,A -85,B 0,C 180,E1 2285.196,E2 2285.196} C_VEL
LIN {X 0,Y 577.8,Z 526.81,A -85,B 0,C 180,E1 2290.923,E2 2290.923} C_VEL
LIN {X 0,Y 577.962,Z 526.81,A -85,B 0,C 180,E1 2297.176,E2 2297.176} C_VEL
LIN {X 0,Y 577.936,Z 526.81,A -85,B 0,C 180,E1 2302.944,E2 2302.944} C_VEL
LIN {X 0,Y 577.916,Z 526.81,A -85,B 0,C 180,E1 2308.397,E2 2308.397} C_VEL
LIN {X 0,Y 577.976,Z 526.81,A -85,B 0,C 180,E1 2313.552,E2 2313.552} C_VEL
LIN {X 0,Y 578.057,Z 526.81,A -85,B 0,C 180,E1 2318.484,E2 2318.484} C_VEL
LIN {X 0,Y 578.228,Z 526.81,A -85,B 0,C 180,E1 2323.256,E2 2323.256} C_VEL
LIN {X 0,Y 578.185,Z 526.81,A -85,B 0,C 180,E1 2329.433,E2 2329.433} C_VEL
LIN {X 0,Y 578.377,Z 526.81,A -85,B 0,C 180,E1 2334.096,E2 2334.096} C_VEL
LIN {X 0,Y 578.173,Z 526.81,A -85,B 0,C 180,E1 2339.995,E2 2339.995} C_VEL
LIN {X 0,Y 578.234,Z 526.81,A -85,B 0,C 180,E1 2344.501,E2 2344.501} C_VEL
LIN {X 0,Y 578.137,Z 526.81,A -85,B 0,C 180,E1 2347.778,E2 2347.778} C_VEL
LIN {X 0,Y 576.824,Z 526.81,A -85,B 0,C 180,E1 2348.633,E2 2348.633} C_VEL
LIN {X 0,Y 570.174,Z 526.81,A -85,B 0,C 180,E1 2350.959,E2 2350.959} C_VEL
LIN {X 0,Y 570.084,Z 526.81,A -85,B 0,C 180,E1 2351.179,E2 2351.179} C_VEL
LIN {X 0,Y 570.064,Z 526.81,A -85,B 0,C 180,E1 2355.397,E2 2355.397} C_VEL
LIN {X 0,Y 570.084,Z 526.81,A -85,B 0,C 180,E1 2360.192,E2 2360.192} C_VEL
LIN {X 0,Y 569.98,Z 526.81,A -85,B 0,C 180,E1 2365.432,E2 2365.432} C_VEL
LIN {X 0,Y 569.975,Z 526.81,A -85,B 0,C 180,E1 2370.305,E2 2370.305} C_VEL
LIN {X 0,Y 570.097,Z 526.81,A -85,B 0,C 180,E1 2375.744,E2 2375.744} C_VEL
LIN {X 0,Y 569.872,Z 526.81,A -85,B 0,C 180,E1 2381.939,E2 2381.939} C_VEL
LIN {X 0,Y 569.837,Z 526.81,A -85,B 0,C 180,E1 2388.38,E2 2388.38} C_VEL
LIN {X 0,Y 569.944,Z 526.81,A -85,B 0,C 180,E1 2394.241,E2 2394.241} C_VEL
LIN {X 0,Y 569.996,Z 526.81,A -85,B 0,C 180,E1 2399.693,E2 2399.693} C_VEL
LIN {X 0,Y 570.151,Z 526.81,A -85,B 0,C 180,E1 2404.86,E2 2404.86} C_VEL
LIN {X 0,Y 570.256,Z 526.81,A -85,B 0,C 180,E1 2407.426,E2 2407.426} C_VEL
LIN {X 0,Y 573.516,Z 540.954,A -85,B 0,C 180,E1 2407.761,E2 2407.761} C_VEL
LIN {X 0,Y 573.495,Z 608.186,A -85,B 0,C 180,E1 2408.769,E2 2408.769} C_VEL
LIN {X 0,Y 573.001,Z 640.646,A -85,B 0,C 180,E1 2409.837,E2 2409.837} C_VEL
LIN {X 0,Y 572.367,Z 672.149,A -85,B 0,C 180,E1 2411.496,E2 2411.496} C_VEL
LIN {X 0,Y 571.762,Z 700.639,A -85,B 0,C 180,E1 2413.662,E2 2413.662} C_VEL
LIN {X 0,Y 571.218,Z 726.288,A -85,B 0,C 180,E1 2416.398,E2 2416.398} C_VEL
LIN {X 0,Y 570.868,Z 746.815,A -85,B 0,C 180,E1 2419.498,E2 2419.498} C_VEL
LIN {X 0,Y 570.7,Z 761.454,A -85,B 0,C 180,E1 2422.764,E2 2422.764} C_VEL
LIN {X 0,Y 570.608,Z 770.615,A -85,B 0,C 180,E1 2426.2,E2 2426.2} C_VEL
LIN {X 0,Y 570.583,Z 773.42,A -85,B 0,C 180,E1 2428.483,E2 2428.483} C_VEL
LIN {X 0,Y 570.549,Z 773.416,A -85,B 0,C 180,E1 2431.524,E2 2431.524} C_VEL
LIN {X 0,Y 570.634,Z 769.063,A -85,B 0,C 180,E1 2434.569,E2 2434.569} C_VEL
LIN {X 0,Y 570.76,Z 758.545,A -85,B 0,C 180,E1 2438.009,E2 2438.009} C_VEL
LIN {X 0,Y 570.945,Z 743.03,A -85,B 0,C 180,E1 2441.17,E2 2441.17} C_VEL
LIN {X 0,Y 571.346,Z 721.578,A -85,B 0,C 180,E1 2444.174,E2 2444.174} C_VEL
LIN {X 0,Y 571.897,Z 696.015,A -85,B 0,C 180,E1 2446.737,E2 2446.737} C_VEL
LIN {X 0,Y 572.483,Z 667.275,A -85,B 0,C 180,E1 2448.808,E2 2448.808} C_VEL
LIN {X 0,Y 573.034,Z 635.911,A -85,B 0,C 180,E1 2450.359,E2 2450.359} C_VEL
LIN {X 0,Y 573.506,Z 600.978,A -85,B 0,C 180,E1 2451.39,E2 2451.39} C_VEL
LIN {X 0,Y 572.848,Z 535.366,A -85,B 0,C 180,E1 2452.341,E2 2452.341} C_VEL
LIN {X 0,Y 570.275,Z 526.81,A -85,B 0,C 180,E1 2452.64,E2 2452.64} C_VEL
LIN {X 0,Y 570.072,Z 526.81,A -85,B 0,C 180,E1 2456.844,E2 2456.844} C_VEL
LIN {X 0,Y 569.902,Z 526.81,A -85,B 0,C 180,E1 2462.1,E2 2462.1} C_VEL
LIN {X 0,Y 570.017,Z 526.81,A -85,B 0,C 180,E1 2467.661,E2 2467.661} C_VEL
LIN {X 0,Y 569.99,Z 526.81,A -85,B 0,C 180,E1 2473.686,E2 2473.686} C_VEL
LIN {X 0,Y 569.879,Z 526.81,A -85,B 0,C 180,E1 2478.387,E2 2478.387} C_VEL
LIN {X 0,Y 569.922,Z 526.81,A -85,B 0,C 180,E1 2484.243,E2 2484.243} C_VEL
LIN {X 0,Y 570.064,Z 526.81,A -85,B 0,C 180,E1 2489.7,E2 2489.7} C_VEL
LIN {X 0,Y 569.977,Z 526.81,A -85,B 0,C 180,E1 2494.855,E2 2494.855} C_VEL
LIN {X 0,Y 570.054,Z 526.81,A -85,B 0,C 180,E1 2499.807,E2 2499.807} C_VEL
LIN {X 0,Y 569.956,Z 526.81,A -85,B 0,C 180,E1 2504.6,E2 2504.6} C_VEL
LIN {X 0,Y 570.312,Z 526.81,A -85,B 0,C 180,E1 2507.159,E2 2507.159} C_VEL
LIN {X 0,Y 571.585,Z 547.856,A -85,B 0,C 180,E1 2507.977,E2 2507.977} C_VEL
LIN {X 0,Y 571.269,Z 571.57,A -85,B 0,C 180,E1 2509.41,E2 2509.41} C_VEL
LIN {X 0,Y 571.001,Z 591.156,A -85,B 0,C 180,E1 2511.235,E2 2511.235} C_VEL
LIN {X 0,Y 570.813,Z 607.289,A -85,B 0,C 180,E1 2513.532,E2 2513.532} C_VEL
LIN {X 0,Y 570.758,Z 617.338,A -85,B 0,C 180,E1 2515.821,E2 2515.821} C_VEL
LIN {X 0,Y 570.658,Z 623.152,A -85,B 0,C 180,E1 2518.484,E2 2518.484} C_VEL
LIN {X 0,Y 570.684,Z 623.996,A -85,B 0,C 180,E1 2520.005,E2 2520.005} C_VEL
LIN {X 0,Y 570.656,Z 621.92,A -85,B 0,C 180,E1 2522.285,E2 2522.285} C_VEL
LIN {X 0,Y 570.773,Z 614.292,A -85,B 0,C 180,E1 2524.912,E2 2524.912} C_VEL
LIN {X 0,Y 570.825,Z 602.07,A -85,B 0,C 180,E1 2527.242,E2 2527.242} C_VEL
LIN {X 0,Y 571.09,Z 584.791,A -85,B 0,C 180,E1 2529.35,E2 2529.35} C_VEL
LIN {X 0,Y 571.375,Z 562.413,A -85,B 0,C 180,E1 2531.136,E2 2531.136} C_VEL
LIN {X 0,Y 571.666,Z 536.992,A -85,B 0,C 180,E1 2532.382,E2 2532.382} C_VEL
LIN {X 0,Y 570.292,Z 526.81,A -85,B 0,C 180,E1 2532.754,E2 2532.754} C_VEL
LIN {X 0,Y 570.232,Z 526.81,A -85,B 0,C 180,E1 2538.584,E2 2538.584} C_VEL
LIN {X 0,Y 570.141,Z 526.81,A -85,B 0,C 180,E1 2543.478,E2 2543.478} C_VEL
LIN {X 0,Y 569.99,Z 526.81,A -85,B 0,C 180,E1 2548.76,E2 2548.76} C_VEL
LIN {X 0,Y 569.951,Z 526.81,A -85,B 0,C 180,E1 2554.556,E2 2554.556} C_VEL
LIN {X 0,Y 569.923,Z 526.81,A -85,B 0,C 180,E1 2559.616,E2 2559.616} C_VEL
LIN {X 0,Y 569.981,Z 526.81,A -85,B 0,C 180,E1 2565.829,E2 2565.829} C_VEL
LIN {X 0,Y 569.983,Z 526.81,A -85,B 0,C 180,E1 2570.388,E2 2570.388} C_VEL
LIN {X 0,Y 569.899,Z 526.81,A -85,B 0,C 180,E1 2576.084,E2 2576.084} C_VEL
LIN {X 0,Y 569.975,Z 526.81,A -85,B 0,C 180,E1 2581.431,E2 2581.431} C_VEL
LIN {X 0,Y 570.087,Z 526.81,A -85,B 0,C 180,E1 2586.519,E2 2586.519} C_VEL
LIN {X 0,Y 570.257,Z 526.81,A -85,B 0,C 180,E1 2591.417,E2 2591.417} C_VEL
LIN {X 0,Y 569.849,Z 526.81,A -85,B 0,C 180,E1 2596.161,E2 2596.161} C_VEL
LIN {X 0,Y 570.161,Z 526.81,A -85,B 0,C 180,E1 2600.828,E2 2600.828} C_VEL
LIN {X 0,Y 570.247,Z 526.81,A -85,B 0,C 180,E1 2605.428,E2 2605.428} C_VEL
LIN {X 0,Y 570.307,Z 526.81,A -85,B 0,C 180,E1 2609.996,E2 2609.996} C_VEL
LIN {X 0,Y 570.333,Z 526.81,A -85,B 0,C 180,E1 2614.564,E2 2614.564} C_VEL
LIN {X 0,Y 570.274,Z 526.81,A -85,B 0,C 180,E1 2619.163,E2 2619.163} C_VEL
LIN {X 0,Y 570.277,Z 526.81,A -85,B 0,C 180,E1 2623.821,E2 2623.821} C_VEL
LIN {X 0,Y 570.224,Z 526.81,A -85,B 0,C 180,E1 2628.576,E2 2628.576} C_VEL
LIN {X 0,Y 570.132,Z 526.81,A -85,B 0,C 180,E1 2633.471,E2 2633.471} C_VEL
LIN {X 0,Y 569.976,Z 526.81,A -85,B 0,C 180,E1 2638.76,E2 2638.76} C_VEL
LIN {X 0,Y 569.946,Z 526.81,A -85,B 0,C 180,E1 2644.557,E2 2644.557} C_VEL
LIN {X 0,Y 569.9,Z 526.81,A -85,B 0,C 180,E1 2649.609,E2 2649.609} C_VEL
LIN {X 0,Y 569.937,Z 526.81,A -85,B 0,C 180,E1 2655.824,E2 2655.824} C_VEL
LIN {X 0,Y 569.981,Z 526.81,A -85,B 0,C 180,E1 2660.389,E2 2660.389} C_VEL
LIN {X 0,Y 569.893,Z 526.81,A -85,B 0,C 180,E1 2666.084,E2 2666.084} C_VEL
LIN {X 0,Y 569.946,Z 526.81,A -85,B 0,C 180,E1 2671.43,E2 2671.43} C_VEL
LIN {X 0,Y 570.076,Z 526.81,A -85,B 0,C 180,E1 2676.519,E2 2676.519} C_VEL
LIN {X 0,Y 570.282,Z 526.81,A -85,B 0,C 180,E1 2681.418,E2 2681.418} C_VEL
LIN {X 0,Y 569.976,Z 526.81,A -85,B 0,C 180,E1 2687.726,E2 2687.726} C_VEL
LIN {X 0,Y 570.44,Z 526.81,A -85,B 0,C 180,E1 2693.901,E2 2693.901} C_VEL
LIN {X 0,Y 570.285,Z 526.81,A -85,B 0,C 180,E1 2699.995,E2 2699.995} C_VEL
LIN {X 0,Y 570.329,Z 526.81,A -85,B 0,C 180,E1 2704.563,E2 2704.563} C_VEL
LIN {X 0,Y 570.244,Z 526.81,A -85,B 0,C 180,E1 2709.161,E2 2709.161} C_VEL
LIN {X 0,Y 570.084,Z 526.81,A -85,B 0,C 180,E1 2711.179,E2 2711.179} C_VEL
LIN {X 0,Y 568.865,Z 526.81,A -85,B 0,C 180,E1 2712.047,E2 2712.047} C_VEL
LIN {X 0,Y 562.191,Z 526.81,A -85,B 0,C 180,E1 2714.633,E2 2714.633} C_VEL
LIN {X 0,Y 562.203,Z 526.81,A -85,B 0,C 180,E1 2719.521,E2 2719.521} C_VEL
LIN {X 0,Y 562.085,Z 526.81,A -85,B 0,C 180,E1 2725.523,E2 2725.523} C_VEL
LIN {X 0,Y 562.076,Z 526.81,A -85,B 0,C 180,E1 2730.777,E2 2730.777} C_VEL
LIN {X 0,Y 562.137,Z 526.81,A -85,B 0,C 180,E1 2736.33,E2 2736.33} C_VEL
LIN {X 0,Y 561.92,Z 526.81,A -85,B 0,C 180,E1 2742.337,E2 2742.337} C_VEL
LIN {X 0,Y 561.894,Z 526.81,A -85,B 0,C 180,E1 2747.656,E2 2747.656} C_VEL
LIN {X 0,Y 562.018,Z 526.81,A -85,B 0,C 180,E1 2753.908,E2 2753.908} C_VEL
LIN {X 0,Y 562.085,Z 526.81,A -85,B 0,C 180,E1 2759.524,E2 2759.524} C_VEL
LIN {X 0,Y 562.256,Z 526.81,A -85,B 0,C 180,E1 2764.482,E2 2764.482} C_VEL
LIN {X 0,Y 562.32,Z 526.81,A -85,B 0,C 180,E1 2767.101,E2 2767.101} C_VEL
LIN {X 0,Y 566.232,Z 541.559,A -85,B 0,C 180,E1 2767.467,E2 2767.467} C_VEL
LIN {X 0,Y 566.148,Z 608.203,A -85,B 0,C 180,E1 2768.481,E2 2768.481} C_VEL
LIN {X 0,Y 565.532,Z 641.288,A -85,B 0,C 180,E1 2769.586,E2 2769.586} C_VEL
LIN {X 0,Y 564.771,Z 673.68,A -85,B 0,C 180,E1 2771.339,E2 2771.339} C_VEL
LIN {X 0,Y 564.004,Z 702.737,A -85,B 0,C 180,E1 2773.632,E2 2773.632} C_VEL
LIN {X 0,Y 563.442,Z 726.287,A -85,B 0,C 180,E1 2776.207,E2 2776.207} C_VEL
LIN {X 0,Y 563.055,Z 745.731,A -85,B 0,C 180,E1 2779.154,E2 2779.154} C_VEL
LIN {X 0,Y 562.88,Z 760.104,A -85,B 0,C 180,E1 2782.274,E2 2782.274} C_VEL
LIN {X 0,Y 562.762,Z 769.077,A -85,B 0,C 180,E1 2785.374,E2 2785.374} C_VEL
LIN {X 0,Y 562.679,Z 773.42,A -85,B 0,C 180,E1 2788.462,E2 2788.462} C_VEL
LIN {X 0,Y 562.646,Z 773.415,A -85,B 0,C 180,E1 2791.546,E2 2791.546} C_VEL
LIN {X 0,Y 562.74,Z 769.062,A -85,B 0,C 180,E1 2794.633,E2 2794.633} C_VEL
LIN {X 0,Y 562.888,Z 758.545,A -85,B 0,C 180,E1 2798.122,E2 2798.122} C_VEL
LIN {X 0,Y 563.127,Z 743.03,A -85,B 0,C 180,E1 2801.327,E2 2801.327} C_VEL
LIN {X 0,Y 563.571,Z 721.478,A -85,B 0,C 180,E1 2804.386,E2 2804.386} C_VEL
LIN {X 0,Y 564.174,Z 696.013,A -85,B 0,C 180,E1 2806.973,E2 2806.973} C_VEL
LIN {X 0,Y 564.923,Z 667.278,A -85,B 0,C 180,E1 2809.069,E2 2809.069} C_VEL
LIN {X 0,Y 565.686,Z 634.443,A -85,B 0,C 180,E1 2810.697,E2 2810.697} C_VEL
LIN {X 0,Y 566.161,Z 599.748,A -85,B 0,C 180,E1 2811.707,E2 2811.707} C_VEL
LIN {X 0,Y 565.689,Z 537.432,A -85,B 0,C 180,E1 2812.611,E2 2812.611} C_VEL
LIN {X 0,Y 562.346,Z 526.81,A -85,B 0,C 180,E1 2812.95,E2 2812.95} C_VEL
LIN {X 0,Y 562.103,Z 526.81,A -85,B 0,C 180,E1 2817.283,E2 2817.283} C_VEL
LIN {X 0,Y 561.932,Z 526.81,A -85,B 0,C 180,E1 2822.612,E2 2822.612} C_VEL
LIN {X 0,Y 562.027,Z 526.81,A -85,B 0,C 180,E1 2828.292,E2 2828.292} C_VEL
LIN {X 0,Y 562.065,Z 526.81,A -85,B 0,C 180,E1 2834.462,E2 2834.462} C_VEL
LIN {X 0,Y 561.933,Z 526.81,A -85,B 0,C 180,E1 2839.719,E2 2839.719} C_VEL
LIN {X 0,Y 562.077,Z 526.81,A -85,B 0,C 180,E1 2845.558,E2 2845.558} C_VEL
LIN {X 0,Y 562.118,Z 526.81,A -85,B 0,C 180,E1 2851.006,E2 2851.006} C_VEL
LIN {X 0,Y 562.14,Z 526.81,A -85,B 0,C 180,E1 2856.322,E2 2856.322} C_VEL
LIN {X 0,Y 562.243,Z 526.81,A -85,B 0,C 180,E1 2861.153,E2 2861.153} C_VEL
LIN {X 0,Y 562.346,Z 526.81,A -85,B 0,C 180,E1 2866.974,E2 2866.974} C_VEL
LIN {X 0,Y 563.864,Z 546.966,A -85,B 0,C 180,E1 2867.769,E2 2867.769} C_VEL
LIN {X 0,Y 563.453,Z 571.559,A -85,B 0,C 180,E1 2869.262,E2 2869.262} C_VEL
LIN {X 0,Y 563.168,Z 591.15,A -85,B 0,C 180,E1 2871.112,E2 2871.112} C_VEL
LIN {X 0,Y 562.935,Z 607.286,A -85,B 0,C 180,E1 2873.441,E2 2873.441} C_VEL
LIN {X 0,Y 562.87,Z 617.336,A -85,B 0,C 180,E1 2875.763,E2 2875.763} C_VEL
LIN {X 0,Y 562.759,Z 623.151,A -85,B 0,C 180,E1 2878.463,E2 2878.463} C_VEL
LIN {X 0,Y 562.784,Z 623.996,A -85,B 0,C 180,E1 2880.005,E2 2880.005} C_VEL
LIN {X 0,Y 562.775,Z 621.921,A -85,B 0,C 180,E1 2882.317,E2 2882.317} C_VEL
LIN {X 0,Y 562.88,Z 614.359,A -85,B 0,C 180,E1 2884.965,E2 2884.965} C_VEL
LIN {X 0,Y 562.961,Z 602.075,A -85,B 0,C 180,E1 2887.344,E2 2887.344} C_VEL
LIN {X 0,Y 563.265,Z 584.796,A -85,B 0,C 180,E1 2889.481,E2 2889.481} C_VEL
LIN {X 0,Y 563.584,Z 564.165,A -85,B 0,C 180,E1 2891.18,E2 2891.18} C_VEL
LIN {X 0,Y 563.943,Z 538.364,A -85,B 0,C 180,E1 2892.505,E2 2892.505} C_VEL
LIN {X 0,Y 562.324,Z 526.81,A -85,B 0,C 180,E1 2892.937,E2 2892.937} C_VEL
LIN {X 0,Y 562.284,Z 526.81,A -85,B 0,C 180,E1 2898.856,E2 2898.856} C_VEL
LIN {X 0,Y 562.191,Z 526.81,A -85,B 0,C 180,E1 2903.831,E2 2903.831} C_VEL
LIN {X 0,Y 562.055,Z 526.81,A -85,B 0,C 180,E1 2909.009,E2 2909.009} C_VEL
LIN {X 0,Y 562.062,Z 526.81,A -85,B 0,C 180,E1 2914.454,E2 2914.454} C_VEL
LIN {X 0,Y 561.926,Z 526.81,A -85,B 0,C 180,E1 2920.294,E2 2920.294} C_VEL
LIN {X 0,Y 562.05,Z 526.81,A -85,B 0,C 180,E1 2925.536,E2 2925.536} C_VEL
LIN {X 0,Y 562.038,Z 526.81,A -85,B 0,C 180,E1 2931.709,E2 2931.709} C_VEL
LIN {X 0,Y 561.99,Z 526.81,A -85,B 0,C 180,E1 2937.392,E2 2937.392} C_VEL
LIN {X 0,Y 562.129,Z 526.81,A -85,B 0,C 180,E1 2942.745,E2 2942.745} C_VEL
LIN {X 0,Y 562.16,Z 526.81,A -85,B 0,C 180,E1 2947.844,E2 2947.844} C_VEL
LIN {X 0,Y 562.369,Z 526.81,A -85,B 0,C 180,E1 2952.769,E2 2952.769} C_VEL
LIN {X 0,Y 562.321,Z 526.81,A -85,B 0,C 180,E1 2959.132,E2 2959.132} C_VEL
LIN {X 0,Y 562.379,Z 526.81,A -85,B 0,C 180,E1 2964.982,E2 2964.982} C_VEL
LIN {X 0,Y 562.407,Z 526.81,A -85,B 0,C 180,E1 2969.996,E2 2969.996} C_VEL
LIN {X 0,Y 562.353,Z 526.81,A -85,B 0,C 180,E1 2974.988,E2 2974.988} C_VEL
LIN {X 0,Y 562.366,Z 526.81,A -85,B 0,C 180,E1 2979.293,E2 2979.293} C_VEL
LIN {X 0,Y 562.299,Z 526.81,A -85,B 0,C 180,E1 2984.215,E2 2984.215} C_VEL
LIN {X 0,Y 562.233,Z 526.81,A -85,B 0,C 180,E1 2989.513,E2 2989.513} C_VEL
LIN {X 0,Y 562.084,Z 526.81,A -85,B 0,C 180,E1 2995.526,E2 2995.526} C_VEL
LIN {X 0,Y 562.025,Z 526.81,A -85,B 0,C 180,E1 3000.783,E2 3000.783} C_VEL
LIN {X 0,Y 561.998,Z 526.81,A -85,B 0,C 180,E1 3006.344,E2 3006.344} C_VEL
LIN {X 0,Y 561.913,Z 526.81,A -85,B 0,C 180,E1 3012.342,E2 3012.342} C_VEL
LIN {X 0,Y 562.032,Z 526.81,A -85,B 0,C 180,E1 3017.66,E2 3017.66} C_VEL
LIN {X 0,Y 562.066,Z 526.81,A -85,B 0,C 180,E1 3023.907,E2 3023.907} C_VEL
LIN {X 0,Y 562.117,Z 526.81,A -85,B 0,C 180,E1 3029.526,E2 3029.526} C_VEL
LIN {X 0,Y 562.207,Z 526.81,A -85,B 0,C 180,E1 3034.472,E2 3034.472} C_VEL
LIN {X 0,Y 562.319,Z 526.81,A -85,B 0,C 180,E1 3040.446,E2 3040.446} C_VEL
LIN {X 0,Y 562.162,Z 526.81,A -85,B 0,C 180,E1 3044.372,E2 3044.372} C_VEL
LIN {X 0,Y 562.276,Z 526.81,A -85,B 0,C 180,E1 3050.698,E2 3050.698} C_VEL
LIN {X 0,Y 562.341,Z 526.81,A -85,B 0,C 180,E1 3055.362,E2 3055.362} C_VEL
LIN {X 0,Y 562.384,Z 526.81,A -85,B 0,C 180,E1 3059.995,E2 3059.995} C_VEL
LIN {X 0,Y 562.343,Z 526.81,A -85,B 0,C 180,E1 3065.041,E2 3065.041} C_VEL
LIN {X 0,Y 562.19,Z 526.81,A -85,B 0,C 180,E1 3070.861,E2 3070.861} C_VEL
LIN {X 0,Y 562.191,Z 526.81,A -85,B 0,C 180,E1 3074.633,E2 3074.633} C_VEL
LIN {X 0,Y 558.207,Z 526.81,A -85,B 0,C 180,E1 3076.377,E2 3076.377} C_VEL
LIN {X 0,Y 554.285,Z 526.81,A -85,B 0,C 180,E1 3078.146,E2 3078.146} C_VEL
LIN {X 0,Y 554.193,Z 526.81,A -85,B 0,C 180,E1 3084.186,E2 3084.186} C_VEL
LIN {X 0,Y 554.163,Z 526.81,A -85,B 0,C 180,E1 3089.451,E2 3089.451} C_VEL
LIN {X 0,Y 554.259,Z 526.81,A -85,B 0,C 180,E1 3094.998,E2 3094.998} C_VEL
LIN {X 0,Y 554.056,Z 526.81,A -85,B 0,C 180,E1 3100.975,E2 3100.975} C_VEL
LIN {X 0,Y 554.003,Z 526.81,A -85,B 0,C 180,E1 3107.542,E2 3107.542} C_VEL
LIN {X 0,Y 553.993,Z 526.81,A -85,B 0,C 180,E1 3113.044,E2 3113.044} C_VEL
LIN {X 0,Y 554.069,Z 526.81,A -85,B 0,C 180,E1 3118.726,E2 3118.726} C_VEL
LIN {X 0,Y 554.322,Z 526.81,A -85,B 0,C 180,E1 3124.32,E2 3124.32} C_VEL
LIN {X 0,Y 554.392,Z 526.81,A -85,B 0,C 180,E1 3126.727,E2 3126.727} C_VEL
LIN {X 0,Y 558.933,Z 541.798,A -85,B 0,C 180,E1 3127.16,E2 3127.16} C_VEL
LIN {X 0,Y 558.819,Z 608.185,A -85,B 0,C 180,E1 3128.184,E2 3128.184} C_VEL
LIN {X 0,Y 558.07,Z 642.483,A -85,B 0,C 180,E1 3129.352,E2 3129.352} C_VEL
LIN {X 0,Y 557.178,Z 674.613,A -85,B 0,C 180,E1 3131.138,E2 3131.138} C_VEL
LIN {X 0,Y 556.319,Z 702.735,A -85,B 0,C 180,E1 3133.399,E2 3133.399} C_VEL
LIN {X 0,Y 555.637,Z 727.784,A -85,B 0,C 180,E1 3136.21,E2 3136.21} C_VEL
LIN {X 0,Y 555.16,Z 747.896,A -85,B 0,C 180,E1 3139.396,E2 3139.396} C_VEL
LIN {X 0,Y 554.971,Z 761.455,A -85,B 0,C 180,E1 3142.558,E2 3142.558} C_VEL
LIN {X 0,Y 554.847,Z 770.614,A -85,B 0,C 180,E1 3146.092,E2 3146.092} C_VEL
LIN {X 0,Y 554.775,Z 773.419,A -85,B 0,C 180,E1 3148.44,E2 3148.44} C_VEL
LIN {X 0,Y 554.743,Z 773.415,A -85,B 0,C 180,E1 3151.568,E2 3151.568} C_VEL
LIN {X 0,Y 554.893,Z 767.993,A -85,B 0,C 180,E1 3155.178,E2 3155.178} C_VEL
LIN {X 0,Y 555.011,Z 757.011,A -85,B 0,C 180,E1 3158.633,E2 3158.633} C_VEL
LIN {X 0,Y 555.347,Z 739.929,A -85,B 0,C 180,E1 3162.002,E2 3162.002} C_VEL
LIN {X 0,Y 555.892,Z 718.129,A -85,B 0,C 180,E1 3164.986,E2 3164.986} C_VEL
LIN {X 0,Y 556.673,Z 691.887,A -85,B 0,C 180,E1 3167.568,E2 3167.568} C_VEL
LIN {X 0,Y 557.608,Z 661.381,A -85,B 0,C 180,E1 3169.686,E2 3169.686} C_VEL
LIN {X 0,Y 558.409,Z 629.618,A -85,B 0,C 180,E1 3171.163,E2 3171.163} C_VEL
LIN {X 0,Y 558.855,Z 595.921,A -85,B 0,C 180,E1 3172.084,E2 3172.084} C_VEL
LIN {X 0,Y 558.154,Z 538.587,A -85,B 0,C 180,E1 3172.918,E2 3172.918} C_VEL
LIN {X 0,Y 554.411,Z 526.81,A -85,B 0,C 180,E1 3173.321,E2 3173.321} C_VEL
LIN {X 0,Y 554.136,Z 526.81,A -85,B 0,C 180,E1 3179.049,E2 3179.049} C_VEL
LIN {X 0,Y 554.07,Z 526.81,A -85,B 0,C 180,E1 3185.024,E2 3185.024} C_VEL
LIN {X 0,Y 554.111,Z 526.81,A -85,B 0,C 180,E1 3190.984,E2 3190.984} C_VEL
LIN {X 0,Y 554.078,Z 526.81,A -85,B 0,C 180,E1 3196.919,E2 3196.919} C_VEL
LIN {X 0,Y 554.018,Z 526.81,A -85,B 0,C 180,E1 3203.05,E2 3203.05} C_VEL
LIN {X 0,Y 554.193,Z 526.81,A -85,B 0,C 180,E1 3208.737,E2 3208.737} C_VEL
LIN {X 0,Y 554.148,Z 526.81,A -85,B 0,C 180,E1 3214.383,E2 3214.383} C_VEL
LIN {X 0,Y 554.197,Z 526.81,A -85,B 0,C 180,E1 3219.203,E2 3219.203} C_VEL
LIN {X 0,Y 554.162,Z 526.81,A -85,B 0,C 180,E1 3224.15,E2 3224.15} C_VEL
LIN {X 0,Y 554.415,Z 526.81,A -85,B 0,C 180,E1 3226.784,E2 3226.784} C_VEL
LIN {X 0,Y 556.099,Z 546.422,A -85,B 0,C 180,E1 3227.571,E2 3227.571} C_VEL
LIN {X 0,Y 555.692,Z 570.285,A -85,B 0,C 180,E1 3229.01,E2 3229.01} C_VEL
LIN {X 0,Y 555.327,Z 591.145,A -85,B 0,C 180,E1 3230.986,E2 3230.986} C_VEL
LIN {X 0,Y 555.051,Z 607.282,A -85,B 0,C 180,E1 3233.348,E2 3233.348} C_VEL
LIN {X 0,Y 554.973,Z 618.509,A -85,B 0,C 180,E1 3236.094,E2 3236.094} C_VEL
LIN {X 0,Y 554.859,Z 623.15,A -85,B 0,C 180,E1 3238.441,E2 3238.441} C_VEL
LIN {X 0,Y 554.912,Z 623.996,A -85,B 0,C 180,E1 3240.005,E2 3240.005} C_VEL
LIN {X 0,Y 554.873,Z 621.922,A -85,B 0,C 180,E1 3242.35,E2 3242.35} C_VEL
LIN {X 0,Y 554.999,Z 613.793,A -85,B 0,C 180,E1 3245.181,E2 3245.181} C_VEL
LIN {X 0,Y 555.16,Z 600.765,A -85,B 0,C 180,E1 3247.645,E2 3247.645} C_VEL
LIN {X 0,Y 555.455,Z 582.862,A -85,B 0,C 180,E1 3249.813,E2 3249.813} C_VEL
LIN {X 0,Y 555.887,Z 559.669,A -85,B 0,C 180,E1 3251.629,E2 3251.629} C_VEL
LIN {X 0,Y 555.831,Z 534.344,A -85,B 0,C 180,E1 3252.837,E2 3252.837} C_VEL
LIN {X 0,Y 554.372,Z 526.81,A -85,B 0,C 180,E1 3253.119,E2 3253.119} C_VEL
LIN {X 0,Y 554.35,Z 526.81,A -85,B 0,C 180,E1 3259.136,E2 3259.136} C_VEL
LIN {X 0,Y 554.23,Z 526.81,A -85,B 0,C 180,E1 3264.195,E2 3264.195} C_VEL
LIN {X 0,Y 554.121,Z 526.81,A -85,B 0,C 180,E1 3269.465,E2 3269.465} C_VEL
LIN {X 0,Y 554.098,Z 526.81,A -85,B 0,C 180,E1 3275.021,E2 3275.021} C_VEL
LIN {X 0,Y 554.037,Z 526.81,A -85,B 0,C 180,E1 3280.989,E2 3280.989} C_VEL
LIN {X 0,Y 554.165,Z 526.81,A -85,B 0,C 180,E1 3286.913,E2 3286.913} C_VEL
LIN {X 0,Y 554.107,Z 526.81,A -85,B 0,C 180,E1 3293.044,E2 3293.044} C_VEL
LIN {X 0,Y 554.112,Z 526.81,A -85,B 0,C 180,E1 3298.72,E2 3298.72} C_VEL
LIN {X 0,Y 554.296,Z 526.81,A -85,B 0,C 180,E1 3304.348,E2 3304.348} C_VEL
LIN {X 0,Y 554.407,Z 526.81,A -85,B 0,C 180,E1 3310.866,E2 3310.866} C_VEL
LIN {X 0,Y 554.083,Z 526.81,A -85,B 0,C 180,E1 3315.759,E2 3315.759} C_VEL
LIN {X 0,Y 554.365,Z 526.81,A -85,B 0,C 180,E1 3320.565,E2 3320.565} C_VEL
LIN {X 0,Y 554.473,Z 526.81,A -85,B 0,C 180,E1 3325.297,E2 3325.297} C_VEL
LIN {X 0,Y 554.506,Z 526.81,A -85,B 0,C 180,E1 3329.996,E2 3329.996} C_VEL
LIN {X 0,Y 554.52,Z 526.81,A -85,B 0,C 180,E1 3334.695,E2 3334.695} C_VEL
LIN {X 0,Y 554.351,Z 526.81,A -85,B 0,C 180,E1 3340.492,E2 3340.492} C_VEL
LIN {X 0,Y 554.274,Z 526.81,A -85,B 0,C 180,E1 3345.849,E2 3345.849} C_VEL
LIN {X 0,Y 554.286,Z 526.81,A -85,B 0,C 180,E1 3350.796,E2 3350.796} C_VEL
LIN {X 0,Y 554.136,Z 526.81,A -85,B 0,C 180,E1 3355.919,E2 3355.919} C_VEL
LIN {X 0,Y 554.078,Z 526.81,A -85,B 0,C 180,E1 3361.274,E2 3361.274} C_VEL
LIN {X 0,Y 554.007,Z 526.81,A -85,B 0,C 180,E1 3366.955,E2 3366.955} C_VEL
LIN {X 0,Y 554.027,Z 526.81,A -85,B 0,C 180,E1 3373.09,E2 3373.09} C_VEL
LIN {X 0,Y 554.115,Z 526.81,A -85,B 0,C 180,E1 3379.018,E2 3379.018} C_VEL
LIN {X 0,Y 554.09,Z 526.81,A -85,B 0,C 180,E1 3385.054,E2 3385.054} C_VEL
LIN {X 0,Y 554.164,Z 526.81,A -85,B 0,C 180,E1 3390.954,E2 3390.954} C_VEL
LIN {X 0,Y 554.238,Z 526.81,A -85,B 0,C 180,E1 3395.806,E2 3395.806} C_VEL
LIN {X 0,Y 554.422,Z 526.81,A -85,B 0,C 180,E1 3400.866,E2 3400.866} C_VEL
LIN {X 0,Y 554.122,Z 526.81,A -85,B 0,C 180,E1 3405.76,E2 3405.76} C_VEL
LIN {X 0,Y 554.364,Z 526.81,A -85,B 0,C 180,E1 3410.564,E2 3410.564} C_VEL
LIN {X 0,Y 554.461,Z 526.81,A -85,B 0,C 180,E1 3415.296,E2 3415.296} C_VEL
LIN {X 0,Y 554.484,Z 526.81,A -85,B 0,C 180,E1 3419.995,E2 3419.995} C_VEL
LIN {X 0,Y 554.514,Z 526.81,A -85,B 0,C 180,E1 3424.693,E2 3424.693} C_VEL
LIN {X 0,Y 554.3,Z 526.81,A -85,B 0,C 180,E1 3430.495,E2 3430.495} C_VEL
LIN {X 0,Y 554.246,Z 526.81,A -85,B 0,C 180,E1 3435.848,E2 3435.848} C_VEL
LIN {X 0,Y 554.285,Z 526.81,A -85,B 0,C 180,E1 3438.146,E2 3438.146} C_VEL
LIN {X 0,Y 553.015,Z 526.81,A -85,B 0,C 180,E1 3439.039,E2 3439.039} C_VEL
LIN {X 0,Y 546.375,Z 526.81,A -85,B 0,C 180,E1 3441.468,E2 3441.468} C_VEL
LIN {X 0,Y 546.266,Z 526.81,A -85,B 0,C 180,E1 3441.698,E2 3441.698} C_VEL
LIN {X 0,Y 546.282,Z 526.81,A -85,B 0,C 180,E1 3447.521,E2 3447.521} C_VEL
LIN {X 0,Y 546.291,Z 526.81,A -85,B 0,C 180,E1 3453.758,E2 3453.758} C_VEL
LIN {X 0,Y 546.168,Z 526.81,A -85,B 0,C 180,E1 3459.604,E2 3459.604} C_VEL
LIN {X 0,Y 546.004,Z 526.81,A -85,B 0,C 180,E1 3466.125,E2 3466.125} C_VEL
LIN {X 0,Y 546.037,Z 526.81,A -85,B 0,C 180,E1 3470.92,E2 3470.92} C_VEL
LIN {X 0,Y 546.079,Z 526.81,A -85,B 0,C 180,E1 3476.327,E2 3476.327} C_VEL
LIN {X 0,Y 546.275,Z 526.81,A -85,B 0,C 180,E1 3482.472,E2 3482.472} C_VEL
LIN {X 0,Y 546.481,Z 526.81,A -85,B 0,C 180,E1 3486.419,E2 3486.419} C_VEL
LIN {X 0,Y 551.684,Z 544.585,A -85,B 0,C 180,E1 3486.881,E2 3486.881} C_VEL
LIN {X 0,Y 551.494,Z 608.293,A -85,B 0,C 180,E1 3487.882,E2 3487.882} C_VEL
LIN {X 0,Y 550.683,Z 641.333,A -85,B 0,C 180,E1 3489.011,E2 3489.011} C_VEL
LIN {X 0,Y 549.674,Z 673.208,A -85,B 0,C 180,E1 3490.775,E2 3490.775} C_VEL
LIN {X 0,Y 548.702,Z 701.684,A -85,B 0,C 180,E1 3493.059,E2 3493.059} C_VEL
LIN {X 0,Y 547.892,Z 726.285,A -85,B 0,C 180,E1 3495.807,E2 3495.807} C_VEL
LIN {X 0,Y 547.358,Z 746.601,A -85,B 0,C 180,E1 3499.002,E2 3499.002} C_VEL
LIN {X 0,Y 547.084,Z 761.455,A -85,B 0,C 180,E1 3502.45,E2 3502.45} C_VEL
LIN {X 0,Y 546.947,Z 770.614,A -85,B 0,C 180,E1 3506.035,E2 3506.035} C_VEL
LIN {X 0,Y 546.872,Z 773.419,A -85,B 0,C 180,E1 3508.417,E2 3508.417} C_VEL
LIN {X 0,Y 546.841,Z 773.415,A -85,B 0,C 180,E1 3511.59,E2 3511.59} C_VEL
LIN {X 0,Y 546.975,Z 768.831,A -85,B 0,C 180,E1 3514.884,E2 3514.884} C_VEL
LIN {X 0,Y 547.123,Z 758.544,A -85,B 0,C 180,E1 3518.358,E2 3518.358} C_VEL
LIN {X 0,Y 547.468,Z 742.335,A -85,B 0,C 180,E1 3521.773,E2 3521.773} C_VEL
LIN {X 0,Y 548.073,Z 721.367,A -85,B 0,C 180,E1 3524.816,E2 3524.816} C_VEL
LIN {X 0,Y 548.911,Z 696.008,A -85,B 0,C 180,E1 3527.459,E2 3527.459} C_VEL
LIN {X 0,Y 549.924,Z 666.221,A -85,B 0,C 180,E1 3529.675,E2 3529.675} C_VEL
LIN {X 0,Y 550.884,Z 634.211,A -85,B 0,C 180,E1 3531.29,E2 3531.29} C_VEL
LIN {X 0,Y 551.514,Z 599.342,A -85,B 0,C 180,E1 3532.323,E2 3532.323} C_VEL
LIN {X 0,Y 551.086,Z 540.993,A -85,B 0,C 180,E1 3533.195,E2 3533.195} C_VEL
LIN {X 0,Y 546.513,Z 526.81,A -85,B 0,C 180,E1 3533.604,E2 3533.604} C_VEL
LIN {X 0,Y 546.148,Z 526.81,A -85,B 0,C 180,E1 3539.939,E2 3539.939} C_VEL
LIN {X 0,Y 546.11,Z 526.81,A -85,B 0,C 180,E1 3545.611,E2 3545.611} C_VEL
LIN {X 0,Y 546.211,Z 526.81,A -85,B 0,C 180,E1 3551.708,E2 3551.708} C_VEL
LIN {X 0,Y 546.167,Z 526.81,A -85,B 0,C 180,E1 3556.138,E2 3556.138} C_VEL
LIN {X 0,Y 546.119,Z 526.81,A -85,B 0,C 180,E1 3562.424,E2 3562.424} C_VEL
LIN {X 0,Y 546.279,Z 526.81,A -85,B 0,C 180,E1 3568.231,E2 3568.231} C_VEL
LIN {X 0,Y 546.17,Z 526.81,A -85,B 0,C 180,E1 3573.677,E2 3573.677} C_VEL
LIN {X 0,Y 546.274,Z 526.81,A -85,B 0,C 180,E1 3578.887,E2 3578.887} C_VEL
LIN {X 0,Y 546.279,Z 526.81,A -85,B 0,C 180,E1 3583.915,E2 3583.915} C_VEL
LIN {X 0,Y 546.485,Z 526.954,A -85,B 0,C 180,E1 3586.6,E2 3586.6} C_VEL
LIN {X 0,Y 548.388,Z 545.412,A -85,B 0,C 180,E1 3587.347,E2 3587.347} C_VEL
LIN {X 0,Y 547.917,Z 570.275,A -85,B 0,C 180,E1 3588.852,E2 3588.852} C_VEL
LIN {X 0,Y 547.497,Z 591.14,A -85,B 0,C 180,E1 3590.856,E2 3590.856} C_VEL
LIN {X 0,Y 547.177,Z 607.278,A -85,B 0,C 180,E1 3593.252,E2 3593.252} C_VEL
LIN {X 0,Y 547.078,Z 616.719,A -85,B 0,C 180,E1 3595.457,E2 3595.457} C_VEL
LIN {X 0,Y 547.003,Z 622.078,A -85,B 0,C 180,E1 3597.625,E2 3597.625} C_VEL
LIN {X 0,Y 547.011,Z 623.996,A -85,B 0,C 180,E1 3600.005,E2 3600.005} C_VEL
LIN {X 0,Y 546.981,Z 621.922,A -85,B 0,C 180,E1 3602.384,E2 3602.384} C_VEL
LIN {X 0,Y 547.118,Z 614.302,A -85,B 0,C 180,E1 3605.125,E2 3605.125} C_VEL
LIN {X 0,Y 547.289,Z 600.769,A -85,B 0,C 180,E1 3607.755,E2 3607.755} C_VEL
LIN {X 0,Y 547.647,Z 582.869,A -85,B 0,C 180,E1 3609.955,E2 3609.955} C_VEL
LIN {X 0,Y 548.116,Z 560.219,A -85,B 0,C 180,E1 3611.761,E2 3611.761} C_VEL
LIN {X 0,Y 547.963,Z 534.879,A -85,B 0,C 180,E1 3613.006,E2 3613.006} C_VEL
LIN {X 0,Y 546.423,Z 526.81,A -85,B 0,C 180,E1 3613.353,E2 3613.353} C_VEL
LIN {X 0,Y 546.421,Z 526.81,A -85,B 0,C 180,E1 3619.582,E2 3619.582} C_VEL
LIN {X 0,Y 546.316,Z 526.81,A -85,B 0,C 180,E1 3624.568,E2 3624.568} C_VEL
LIN {X 0,Y 546.146,Z 526.81,A -85,B 0,C 180,E1 3630.743,E2 3630.743} C_VEL
LIN {X 0,Y 546.079,Z 526.81,A -85,B 0,C 180,E1 3636.474,E2 3636.474} C_VEL
LIN {X 0,Y 546.109,Z 526.81,A -85,B 0,C 180,E1 3641.716,E2 3641.716} C_VEL
LIN {X 0,Y 546.208,Z 526.81,A -85,B 0,C 180,E1 3646.128,E2 3646.128} C_VEL
LIN {X 0,Y 546.206,Z 526.81,A -85,B 0,C 180,E1 3652.418,E2 3652.418} C_VEL
LIN {X 0,Y 546.186,Z 526.81,A -85,B 0,C 180,E1 3658.213,E2 3658.213} C_VEL
LIN {X 0,Y 546.29,Z 526.81,A -85,B 0,C 180,E1 3663.672,E2 3663.672} C_VEL
LIN {X 0,Y 546.419,Z 526.81,A -85,B 0,C 180,E1 3668.883,E2 3668.883} C_VEL
LIN {X 0,Y 546.383,Z 526.81,A -85,B 0,C 180,E1 3673.908,E2 3673.908} C_VEL
LIN {X 0,Y 546.468,Z 526.81,A -85,B 0,C 180,E1 3680.427,E2 3680.427} C_VEL
LIN {X 0,Y 546.602,Z 526.81,A -85,B 0,C 180,E1 3685.23,E2 3685.23} C_VEL
LIN {X 0,Y 546.606,Z 526.81,A -85,B 0,C 180,E1 3689.996,E2 3689.996} C_VEL
LIN {X 0,Y 546.619,Z 526.81,A -85,B 0,C 180,E1 3694.763,E2 3694.763} C_VEL
LIN {X 0,Y 546.523,Z 526.81,A -85,B 0,C 180,E1 3699.564,E2 3699.564} C_VEL
LIN {X 0,Y 546.48,Z 526.81,A -85,B 0,C 180,E1 3704.435,E2 3704.435} C_VEL
LIN {X 0,Y 546.415,Z 526.81,A -85,B 0,C 180,E1 3709.585,E2 3709.585} C_VEL
LIN {X 0,Y 546.302,Z 526.81,A -85,B 0,C 180,E1 3714.561,E2 3714.561} C_VEL
LIN {X 0,Y 546.145,Z 526.81,A -85,B 0,C 180,E1 3719.93,E2 3719.93} C_VEL
LIN {X 0,Y 546.104,Z 526.81,A -85,B 0,C 180,E1 3725.602,E2 3725.602} C_VEL
LIN {X 0,Y 546.104,Z 526.81,A -85,B 0,C 180,E1 3731.708,E2 3731.708} C_VEL
LIN {X 0,Y 546.18,Z 526.81,A -85,B 0,C 180,E1 3736.126,E2 3736.126} C_VEL
LIN {X 0,Y 546.182,Z 526.81,A -85,B 0,C 180,E1 3742.417,E2 3742.417} C_VEL
LIN {X 0,Y 546.181,Z 526.81,A -85,B 0,C 180,E1 3748.213,E2 3748.213} C_VEL
LIN {X 0,Y 546.289,Z 526.81,A -85,B 0,C 180,E1 3753.672,E2 3753.672} C_VEL
LIN {X 0,Y 546.418,Z 526.81,A -85,B 0,C 180,E1 3758.882,E2 3758.882} C_VEL
LIN {X 0,Y 546.413,Z 526.81,A -85,B 0,C 180,E1 3763.909,E2 3763.909} C_VEL
LIN {X 0,Y 546.464,Z 526.81,A -85,B 0,C 180,E1 3770.426,E2 3770.426} C_VEL
LIN {X 0,Y 546.517,Z 526.81,A -85,B 0,C 180,E1 3775.769,E2 3775.769} C_VEL
LIN {X 0,Y 546.583,Z 526.81,A -85,B 0,C 180,E1 3779.995,E2 3779.995} C_VEL
LIN {X 0,Y 546.597,Z 526.81,A -85,B 0,C 180,E1 3784.762,E2 3784.762} C_VEL
LIN {X 0,Y 546.484,Z 526.81,A -85,B 0,C 180,E1 3789.563,E2 3789.563} C_VEL
LIN {X 0,Y 546.435,Z 526.81,A -85,B 0,C 180,E1 3794.435,E2 3794.435} C_VEL
LIN {X 0,Y 546.386,Z 526.81,A -85,B 0,C 180,E1 3799.594,E2 3799.594} C_VEL
LIN {X 0,Y 546.266,Z 526.81,A -85,B 0,C 180,E1 3801.698,E2 3801.698} C_VEL
LIN {X 0,Y 542.266,Z 526.81,A -85,B 0,C 180,E1 3803.486,E2 3803.486} C_VEL
LIN {X 0,Y 538.287,Z 526.81,A -85,B 0,C 180,E1 3805.299,E2 3805.299} C_VEL
LIN {X 0,Y 538.292,Z 526.81,A -85,B 0,C 180,E1 3810.41,E2 3810.41} C_VEL
LIN {X 0,Y 538.309,Z 526.81,A -85,B 0,C 180,E1 3816.195,E2 3816.195} C_VEL
LIN {X 0,Y 538.08,Z 526.81,A -85,B 0,C 180,E1 3822.47,E2 3822.47} C_VEL
LIN {X 0,Y 538.054,Z 526.81,A -85,B 0,C 180,E1 3827.524,E2 3827.524} C_VEL
LIN {X 0,Y 538.138,Z 526.81,A -85,B 0,C 180,E1 3833.788,E2 3833.788} C_VEL
LIN {X 0,Y 538.245,Z 526.81,A -85,B 0,C 180,E1 3839.584,E2 3839.584} C_VEL
LIN {X 0,Y 538.416,Z 526.81,A -85,B 0,C 180,E1 3845.055,E2 3845.055} C_VEL
LIN {X 0,Y 538.569,Z 526.81,A -85,B 0,C 180,E1 3846.154,E2 3846.154} C_VEL
LIN {X 0,Y 544.227,Z 546.002,A -85,B 0,C 180,E1 3846.627,E2 3846.627} C_VEL
LIN {X 0,Y 544.062,Z 609.146,A -85,B 0,C 180,E1 3847.614,E2 3847.614} C_VEL
LIN {X 0,Y 543.25,Z 642.469,A -85,B 0,C 180,E1 3848.762,E2 3848.762} C_VEL
LIN {X 0,Y 542.143,Z 673.673,A -85,B 0,C 180,E1 3850.53,E2 3850.53} C_VEL
LIN {X 0,Y 540.992,Z 702.732,A -85,B 0,C 180,E1 3852.915,E2 3852.915} C_VEL
LIN {X 0,Y 540.092,Z 727.787,A -85,B 0,C 180,E1 3855.805,E2 3855.805} C_VEL
LIN {X 0,Y 539.508,Z 747.497,A -85,B 0,C 180,E1 3859.009,E2 3859.009} C_VEL
LIN {X 0,Y 539.208,Z 761.455,A -85,B 0,C 180,E1 3862.339,E2 3862.339} C_VEL
LIN {X 0,Y 539.108,Z 769.076,A -85,B 0,C 180,E1 3865.171,E2 3865.171} C_VEL
LIN {X 0,Y 538.981,Z 773.419,A -85,B 0,C 180,E1 3868.394,E2 3868.394} C_VEL
LIN {X 0,Y 538.952,Z 773.414,A -85,B 0,C 180,E1 3871.614,E2 3871.614} C_VEL
LIN {X 0,Y 539.105,Z 769.06,A -85,B 0,C 180,E1 3874.837,E2 3874.837} C_VEL
LIN {X 0,Y 539.266,Z 758.544,A -85,B 0,C 180,E1 3878.48,E2 3878.48} C_VEL
LIN {X 0,Y 539.638,Z 742.334,A -85,B 0,C 180,E1 3881.946,E2 3881.946} C_VEL
LIN {X 0,Y 540.34,Z 721.368,A -85,B 0,C 180,E1 3885.033,E2 3885.033} C_VEL
LIN {X 0,Y 541.291,Z 696.006,A -85,B 0,C 180,E1 3887.713,E2 3887.713} C_VEL
LIN {X 0,Y 542.387,Z 667.074,A -85,B 0,C 180,E1 3889.907,E2 3889.907} C_VEL
LIN {X 0,Y 543.469,Z 634.917,A -85,B 0,C 180,E1 3891.559,E2 3891.559} C_VEL
LIN {X 0,Y 544.068,Z 601.611,A -85,B 0,C 180,E1 3892.557,E2 3892.557} C_VEL
LIN {X 0,Y 543.52,Z 542.62,A -85,B 0,C 180,E1 3893.424,E2 3893.424} C_VEL
LIN {X 0,Y 538.594,Z 526.81,A -85,B 0,C 180,E1 3893.808,E2 3893.808} C_VEL
LIN {X 0,Y 538.223,Z 526.81,A -85,B 0,C 180,E1 3899.317,E2 3899.317} C_VEL
LIN {X 0,Y 538.172,Z 526.81,A -85,B 0,C 180,E1 3905.339,E2 3905.339} C_VEL
LIN {X 0,Y 538.206,Z 526.81,A -85,B 0,C 180,E1 3910.586,E2 3910.586} C_VEL
LIN {X 0,Y 538.213,Z 526.81,A -85,B 0,C 180,E1 3915.319,E2 3915.319} C_VEL
LIN {X 0,Y 538.198,Z 526.81,A -85,B 0,C 180,E1 3921.977,E2 3921.977} C_VEL
LIN {X 0,Y 538.308,Z 526.81,A -85,B 0,C 180,E1 3927.704,E2 3927.704} C_VEL
LIN {X 0,Y 538.254,Z 526.81,A -85,B 0,C 180,E1 3933.259,E2 3933.259} C_VEL
LIN {X 0,Y 538.329,Z 526.81,A -85,B 0,C 180,E1 3938.56,E2 3938.56} C_VEL
LIN {X 0,Y 538.369,Z 526.81,A -85,B 0,C 180,E1 3943.672,E2 3943.672} C_VEL
LIN {X 0,Y 538.562,Z 526.81,A -85,B 0,C 180,E1 3946.344,E2 3946.344} C_VEL
LIN {X 0,Y 540.751,Z 545.333,A -85,B 0,C 180,E1 3947.113,E2 3947.113} C_VEL
LIN {X 0,Y 540.246,Z 569.587,A -85,B 0,C 180,E1 3948.59,E2 3948.59} C_VEL
LIN {X 0,Y 539.737,Z 589.656,A -85,B 0,C 180,E1 3950.52,E2 3950.52} C_VEL
LIN {X 0,Y 539.318,Z 606.189,A -85,B 0,C 180,E1 3952.95,E2 3952.95} C_VEL
LIN {X 0,Y 539.176,Z 617.503,A -85,B 0,C 180,E1 3955.631,E2 3955.631} C_VEL
LIN {X 0,Y 539.074,Z 623.147,A -85,B 0,C 180,E1 3958.396,E2 3958.396} C_VEL
LIN {X 0,Y 539.113,Z 623.996,A -85,B 0,C 180,E1 3960.005,E2 3960.005} C_VEL
LIN {X 0,Y 539.103,Z 621.923,A -85,B 0,C 180,E1 3962.419,E2 3962.419} C_VEL
LIN {X 0,Y 539.227,Z 614.15,A -85,B 0,C 180,E1 3965.241,E2 3965.241} C_VEL
LIN {X 0,Y 539.42,Z 600.773,A -85,B 0,C 180,E1 3967.869,E2 3967.869} C_VEL
LIN {X 0,Y 539.859,Z 583.51,A -85,B 0,C 180,E1 3970.059,E2 3970.059} C_VEL
LIN {X 0,Y 540.406,Z 560.697,A -85,B 0,C 180,E1 3971.929,E2 3971.929} C_VEL
LIN {X 0,Y 540.297,Z 536.155,A -85,B 0,C 180,E1 3973.172,E2 3973.172} C_VEL
LIN {X 0,Y 538.498,Z 526.81,A -85,B 0,C 180,E1 3973.573,E2 3973.573} C_VEL
LIN {X 0,Y 538.513,Z 526.81,A -85,B 0,C 180,E1 3979.722,E2 3979.722} C_VEL
LIN {X 0,Y 538.285,Z 526.81,A -85,B 0,C 180,E1 3985.822,E2 3985.822} C_VEL
LIN {X 0,Y 538.257,Z 526.81,A -85,B 0,C 180,E1 3990.423,E2 3990.423} C_VEL
LIN {X 0,Y 538.173,Z 526.81,A -85,B 0,C 180,E1 3996.218,E2 3996.218} C_VEL
LIN {X 0,Y 538.139,Z 526.81,A -85,B 0,C 180,E1 4002.477,E2 4002.477} C_VEL
LIN {X 0,Y 538.226,Z 526.81,A -85,B 0,C 180,E1 4007.53,E2 4007.53} C_VEL
LIN {X 0,Y 538.234,Z 526.81,A -85,B 0,C 180,E1 4013.786,E2 4013.786} C_VEL
LIN {X 0,Y 538.284,Z 526.81,A -85,B 0,C 180,E1 4019.578,E2 4019.578} C_VEL
LIN {X 0,Y 538.388,Z 526.81,A -85,B 0,C 180,E1 4025.045,E2 4025.045} C_VEL
LIN {X 0,Y 538.558,Z 526.81,A -85,B 0,C 180,E1 4030.28,E2 4030.28} C_VEL
LIN {X 0,Y 538.309,Z 526.81,A -85,B 0,C 180,E1 4035.333,E2 4035.333} C_VEL
LIN {X 0,Y 538.548,Z 526.81,A -85,B 0,C 180,E1 4040.285,E2 4040.285} C_VEL
LIN {X 0,Y 538.699,Z 526.81,A -85,B 0,C 180,E1 4045.159,E2 4045.159} C_VEL
LIN {X 0,Y 538.724,Z 526.81,A -85,B 0,C 180,E1 4049.996,E2 4049.996} C_VEL
LIN {X 0,Y 538.705,Z 526.81,A -85,B 0,C 180,E1 4054.833,E2 4054.833} C_VEL
LIN {X 0,Y 538.534,Z 526.81,A -85,B 0,C 180,E1 4060.248,E2 4060.248} C_VEL
LIN {X 0,Y 538.545,Z 526.81,A -85,B 0,C 180,E1 4064.653,E2 4064.653} C_VEL
LIN {X 0,Y 538.51,Z 526.81,A -85,B 0,C 180,E1 4069.714,E2 4069.714} C_VEL
LIN {X 0,Y 538.294,Z 526.81,A -85,B 0,C 180,E1 4075.828,E2 4075.828} C_VEL
LIN {X 0,Y 538.242,Z 526.81,A -85,B 0,C 180,E1 4080.416,E2 4080.416} C_VEL
LIN {X 0,Y 538.176,Z 526.81,A -85,B 0,C 180,E1 4086.209,E2 4086.209} C_VEL
LIN {X 0,Y 538.118,Z 526.81,A -85,B 0,C 180,E1 4092.47,E2 4092.47} C_VEL
LIN {X 0,Y 538.194,Z 526.81,A -85,B 0,C 180,E1 4097.528,E2 4097.528} C_VEL
LIN {X 0,Y 538.215,Z 526.81,A -85,B 0,C 180,E1 4103.785,E2 4103.785} C_VEL
LIN {X 0,Y 538.277,Z 526.81,A -85,B 0,C 180,E1 4109.578,E2 4109.578} C_VEL
LIN {X 0,Y 538.376,Z 526.81,A -85,B 0,C 180,E1 4115.045,E2 4115.045} C_VEL
LIN {X 0,Y 538.565,Z 526.81,A -85,B 0,C 180,E1 4120.28,E2 4120.28} C_VEL
LIN {X 0,Y 538.326,Z 526.81,A -85,B 0,C 180,E1 4125.333,E2 4125.333} C_VEL
LIN {X 0,Y 538.545,Z 526.81,A -85,B 0,C 180,E1 4130.284,E2 4130.284} C_VEL
LIN {X 0,Y 538.669,Z 526.81,A -85,B 0,C 180,E1 4135.158,E2 4135.158} C_VEL
LIN {X 0,Y 538.7,Z 526.81,A -85,B 0,C 180,E1 4139.995,E2 4139.995} C_VEL
LIN {X 0,Y 538.681,Z 526.81,A -85,B 0,C 180,E1 4144.832,E2 4144.832} C_VEL
LIN {X 0,Y 538.488,Z 526.81,A -85,B 0,C 180,E1 4150.254,E2 4150.254} C_VEL
LIN {X 0,Y 538.502,Z 526.81,A -85,B 0,C 180,E1 4154.652,E2 4154.652} C_VEL
LIN {X 0,Y 538.479,Z 526.81,A -85,B 0,C 180,E1 4159.713,E2 4159.713} C_VEL
LIN {X 0,Y 538.287,Z 526.81,A -85,B 0,C 180,E1 4165.299,E2 4165.299} C_VEL
LIN {X 0,Y 536.994,Z 526.81,A -85,B 0,C 180,E1 4166.222,E2 4166.222} C_VEL
LIN {X 0,Y 530.444,Z 526.81,A -85,B 0,C 180,E1 4168.736,E2 4168.736} C_VEL
LIN {X 0,Y 530.378,Z 526.81,A -85,B 0,C 180,E1 4168.974,E2 4168.974} C_VEL
LIN {X 0,Y 530.414,Z 526.81,A -85,B 0,C 180,E1 4174.805,E2 4174.805} C_VEL
LIN {X 0,Y 530.216,Z 526.81,A -85,B 0,C 180,E1 4181.046,E2 4181.046} C_VEL
LIN {X 0,Y 530.112,Z 526.81,A -85,B 0,C 180,E1 4186.733,E2 4186.733} C_VEL
LIN {X 0,Y 530.177,Z 526.81,A -85,B 0,C 180,E1 4193.156,E2 4193.156} C_VEL
LIN {X 0,Y 530.265,Z 526.81,A -85,B 0,C 180,E1 4199.077,E2 4199.077} C_VEL
LIN {X 0,Y 530.541,Z 526.81,A -85,B 0,C 180,E1 4205.326,E2 4205.326} C_VEL
LIN {X 0,Y 530.62,Z 526.81,A -85,B 0,C 180,E1 4205.868,E2 4205.868} C_VEL
LIN {X 0,Y 536.725,Z 548.358,A -85,B 0,C 180,E1 4206.395,E2 4206.395} C_VEL
LIN {X 0,Y 536.559,Z 607.248,A -85,B 0,C 180,E1 4207.323,E2 4207.323} C_VEL
LIN {X 0,Y 535.697,Z 640.441,A -85,B 0,C 180,E1 4208.447,E2 4208.447} C_VEL
LIN {X 0,Y 534.597,Z 673.21,A -85,B 0,C 180,E1 4210.244,E2 4210.244} C_VEL
LIN {X 0,Y 533.411,Z 700.734,A -85,B 0,C 180,E1 4212.462,E2 4212.462} C_VEL
LIN {X 0,Y 532.387,Z 725.962,A -85,B 0,C 180,E1 4215.342,E2 4215.342} C_VEL
LIN {X 0,Y 531.736,Z 745.728,A -85,B 0,C 180,E1 4218.507,E2 4218.507} C_VEL
LIN {X 0,Y 531.342,Z 760.103,A -85,B 0,C 180,E1 4221.813,E2 4221.813} C_VEL
LIN {X 0,Y 531.208,Z 769.075,A -85,B 0,C 180,E1 4225.099,E2 4225.099} C_VEL
LIN {X 0,Y 531.078,Z 773.418,A -85,B 0,C 180,E1 4228.37,E2 4228.37} C_VEL
LIN {X 0,Y 531.049,Z 773.414,A -85,B 0,C 180,E1 4231.638,E2 4231.638} C_VEL
LIN {X 0,Y 531.209,Z 769.06,A -85,B 0,C 180,E1 4234.909,E2 4234.909} C_VEL
LIN {X 0,Y 531.396,Z 758.544,A -85,B 0,C 180,E1 4238.607,E2 4238.607} C_VEL
LIN {X 0,Y 531.803,Z 742.333,A -85,B 0,C 180,E1 4242.125,E2 4242.125} C_VEL
LIN {X 0,Y 532.61,Z 721.431,A -85,B 0,C 180,E1 4245.248,E2 4245.248} C_VEL
LIN {X 0,Y 533.648,Z 696.087,A -85,B 0,C 180,E1 4247.968,E2 4247.968} C_VEL
LIN {X 0,Y 534.708,Z 669.165,A -85,B 0,C 180,E1 4250.022,E2 4250.022} C_VEL
LIN {X 0,Y 535.765,Z 636.421,A -85,B 0,C 180,E1 4251.702,E2 4251.702} C_VEL
LIN {X 0,Y 536.447,Z 601.73,A -85,B 0,C 180,E1 4252.776,E2 4252.776} C_VEL
LIN {X 0,Y 535.799,Z 543.844,A -85,B 0,C 180,E1 4253.65,E2 4253.65} C_VEL
LIN {X 0,Y 530.669,Z 526.81,A -85,B 0,C 180,E1 4254.096,E2 4254.096} C_VEL
LIN {X 0,Y 530.331,Z 526.81,A -85,B 0,C 180,E1 4259.039,E2 4259.039} C_VEL
LIN {X 0,Y 530.264,Z 526.81,A -85,B 0,C 180,E1 4264.829,E2 4264.829} C_VEL
LIN {X 0,Y 530.286,Z 526.81,A -85,B 0,C 180,E1 4271.053,E2 4271.053} C_VEL
LIN {X 0,Y 530.289,Z 526.81,A -85,B 0,C 180,E1 4276.755,E2 4276.755} C_VEL
LIN {X 0,Y 530.229,Z 526.81,A -85,B 0,C 180,E1 4283.163,E2 4283.163} C_VEL
LIN {X 0,Y 530.377,Z 526.81,A -85,B 0,C 180,E1 4289.087,E2 4289.087} C_VEL
LIN {X 0,Y 530.387,Z 526.81,A -85,B 0,C 180,E1 4294.654,E2 4294.654} C_VEL
LIN {X 0,Y 530.532,Z 526.81,A -85,B 0,C 180,E1 4300.363,E2 4300.363} C_VEL
LIN {X 0,Y 530.62,Z 526.837,A -85,B 0,C 180,E1 4306.099,E2 4306.099} C_VEL
LIN {X 0,Y 533.158,Z 545.484,A -85,B 0,C 180,E1 4306.874,E2 4306.874} C_VEL
LIN {X 0,Y 532.61,Z 570.718,A -85,B 0,C 180,E1 4308.424,E2 4308.424} C_VEL
LIN {X 0,Y 532.06,Z 590.798,A -85,B 0,C 180,E1 4310.382,E2 4310.382} C_VEL
LIN {X 0,Y 531.562,Z 607.259,A -85,B 0,C 180,E1 4312.847,E2 4312.847} C_VEL
LIN {X 0,Y 531.354,Z 618.032,A -85,B 0,C 180,E1 4315.491,E2 4315.491} C_VEL
LIN {X 0,Y 531.198,Z 623.727,A -85,B 0,C 180,E1 4318.372,E2 4318.372} C_VEL
LIN {X 0,Y 531.232,Z 624.53,A -85,B 0,C 180,E1 4320.005,E2 4320.005} C_VEL
LIN {X 0,Y 531.248,Z 622.48,A -85,B 0,C 180,E1 4322.455,E2 4322.455} C_VEL
LIN {X 0,Y 531.402,Z 614.837,A -85,B 0,C 180,E1 4325.318,E2 4325.318} C_VEL
LIN {X 0,Y 531.639,Z 601.648,A -85,B 0,C 180,E1 4327.985,E2 4327.985} C_VEL
LIN {X 0,Y 532.155,Z 583.425,A -85,B 0,C 180,E1 4330.298,E2 4330.298} C_VEL
LIN {X 0,Y 532.715,Z 561.439,A -85,B 0,C 180,E1 4332.104,E2 4332.104} C_VEL
LIN {X 0,Y 532.663,Z 537.52,A -85,B 0,C 180,E1 4333.342,E2 4333.342} C_VEL
LIN {X 0,Y 530.564,Z 526.81,A -85,B 0,C 180,E1 4333.795,E2 4333.795} C_VEL
LIN {X 0,Y 530.563,Z 526.81,A -85,B 0,C 180,E1 4340.03,E2 4340.03} C_VEL
LIN {X 0,Y 530.431,Z 526.81,A -85,B 0,C 180,E1 4345.355,E2 4345.355} C_VEL
LIN {X 0,Y 530.294,Z 526.81,A -85,B 0,C 180,E1 4351.062,E2 4351.062} C_VEL
LIN {X 0,Y 530.221,Z 526.81,A -85,B 0,C 180,E1 4356.906,E2 4356.906} C_VEL
LIN {X 0,Y 530.234,Z 526.81,A -85,B 0,C 180,E1 4363.264,E2 4363.264} C_VEL
LIN {X 0,Y 530.273,Z 526.81,A -85,B 0,C 180,E1 4368.945,E2 4368.945} C_VEL
LIN {X 0,Y 530.3,Z 526.81,A -85,B 0,C 180,E1 4375.174,E2 4375.174} C_VEL
LIN {X 0,Y 530.377,Z 526.81,A -85,B 0,C 180,E1 4380.964,E2 4380.964} C_VEL
LIN {X 0,Y 530.458,Z 526.81,A -85,B 0,C 180,E1 4386.443,E2 4386.443} C_VEL
LIN {X 0,Y 530.641,Z 526.81,A -85,B 0,C 180,E1 4391.704,E2 4391.704} C_VEL
LIN {X 0,Y 530.561,Z 526.81,A -85,B 0,C 180,E1 4398.473,E2 4398.473} C_VEL
LIN {X 0,Y 530.868,Z 526.81,A -85,B 0,C 180,E1 4403.445,E2 4403.445} C_VEL
LIN {X 0,Y 530.824,Z 526.81,A -85,B 0,C 180,E1 4409.996,E2 4409.996} C_VEL
LIN {X 0,Y 530.79,Z 526.81,A -85,B 0,C 180,E1 4414.905,E2 4414.905} C_VEL
LIN {X 0,Y 530.694,Z 526.81,A -85,B 0,C 180,E1 4419.852,E2 4419.852} C_VEL
LIN {X 0,Y 530.628,Z 526.81,A -85,B 0,C 180,E1 4424.876,E2 4424.876} C_VEL
LIN {X 0,Y 530.562,Z 526.81,A -85,B 0,C 180,E1 4430.022,E2 4430.022} C_VEL
LIN {X 0,Y 530.427,Z 526.81,A -85,B 0,C 180,E1 4435.347,E2 4435.347} C_VEL
LIN {X 0,Y 530.282,Z 526.81,A -85,B 0,C 180,E1 4441.062,E2 4441.062} C_VEL
LIN {X 0,Y 530.218,Z 526.81,A -85,B 0,C 180,E1 4446.908,E2 4446.908} C_VEL
LIN {X 0,Y 530.199,Z 526.81,A -85,B 0,C 180,E1 4453.258,E2 4453.258} C_VEL
LIN {X 0,Y 530.281,Z 526.81,A -85,B 0,C 180,E1 4458.947,E2 4458.947} C_VEL
LIN {X 0,Y 530.288,Z 526.81,A -85,B 0,C 180,E1 4465.173,E2 4465.173} C_VEL
LIN {X 0,Y 530.352,Z 526.81,A -85,B 0,C 180,E1 4470.962,E2 4470.962} C_VEL
LIN {X 0,Y 530.45,Z 526.81,A -85,B 0,C 180,E1 4476.442,E2 4476.442} C_VEL
LIN {X 0,Y 530.664,Z 526.81,A -85,B 0,C 180,E1 4481.704,E2 4481.704} C_VEL
LIN {X 0,Y 530.571,Z 526.81,A -85,B 0,C 180,E1 4488.473,E2 4488.473} C_VEL
LIN {X 0,Y 530.842,Z 526.81,A -85,B 0,C 180,E1 4493.444,E2 4493.444} C_VEL
LIN {X 0,Y 530.8,Z 526.81,A -85,B 0,C 180,E1 4499.995,E2 4499.995} C_VEL
LIN {X 0,Y 530.766,Z 526.81,A -85,B 0,C 180,E1 4504.904,E2 4504.904} C_VEL
LIN {X 0,Y 530.651,Z 526.81,A -85,B 0,C 180,E1 4509.852,E2 4509.852} C_VEL
LIN {X 0,Y 530.585,Z 526.81,A -85,B 0,C 180,E1 4514.876,E2 4514.876} C_VEL
LIN {X 0,Y 530.528,Z 526.81,A -85,B 0,C 180,E1 4520.021,E2 4520.021} C_VEL
LIN {X 0,Y 530.409,Z 526.81,A -85,B 0,C 180,E1 4525.345,E2 4525.345} C_VEL
LIN {X 0,Y 530.378,Z 526.81,A -85,B 0,C 180,E1 4528.974,E2 4528.974} C_VEL
LIN {X 0,Y 527.881,Z 526.81,A -85,B 0,C 180,E1 4530.368,E2 4530.368} C_VEL
LIN {X 0,Y 522.541,Z 526.81,A -85,B 0,C 180,E1 4532.457,E2 4532.457} C_VEL
LIN {X 0,Y 522.482,Z 526.81,A -85,B 0,C 180,E1 4532.699,E2 4532.699} C_VEL
LIN {X 0,Y 522.33,Z 526.81,A -85,B 0,C 180,E1 4538.503,E2 4538.503} C_VEL
LIN {X 0,Y 522.194,Z 526.81,A -85,B 0,C 180,E1 4544.086,E2 4544.086} C_VEL
LIN {X 0,Y 522.216,Z 526.81,A -85,B 0,C 180,E1 4550.374,E2 4550.374} C_VEL
LIN {X 0,Y 522.316,Z 526.81,A -85,B 0,C 180,E1 4556.585,E2 4556.585} C_VEL
LIN {X 0,Y 522.479,Z 526.81,A -85,B 0,C 180,E1 4562.381,E2 4562.381} C_VEL
LIN {X 0,Y 522.666,Z 526.826,A -85,B 0,C 180,E1 4565.573,E2 4565.573} C_VEL
LIN {X 0,Y 529.263,Z 550.993,A -85,B 0,C 180,E1 4566.161,E2 4566.161} C_VEL
LIN {X 0,Y 528.975,Z 608.197,A -85,B 0,C 180,E1 4567.097,E2 4567.097} C_VEL
LIN {X 0,Y 528.019,Z 642.326,A -85,B 0,C 180,E1 4568.308,E2 4568.308} C_VEL
LIN {X 0,Y 526.808,Z 674.642,A -85,B 0,C 180,E1 4570.158,E2 4570.158} C_VEL
LIN {X 0,Y 525.611,Z 703.233,A -85,B 0,C 180,E1 4572.521,E2 4572.521} C_VEL
LIN {X 0,Y 524.665,Z 725.961,A -85,B 0,C 180,E1 4575.122,E2 4575.122} C_VEL
LIN {X 0,Y 523.88,Z 745.727,A -85,B 0,C 180,E1 4578.332,E2 4578.332} C_VEL
LIN {X 0,Y 523.464,Z 760.103,A -85,B 0,C 180,E1 4581.689,E2 4581.689} C_VEL
LIN {X 0,Y 523.305,Z 769.075,A -85,B 0,C 180,E1 4585.024,E2 4585.024} C_VEL
LIN {X 0,Y 523.19,Z 773.418,A -85,B 0,C 180,E1 4588.346,E2 4588.346} C_VEL
LIN {X 0,Y 523.163,Z 773.413,A -85,B 0,C 180,E1 4591.662,E2 4591.662} C_VEL
LIN {X 0,Y 523.308,Z 769.059,A -85,B 0,C 180,E1 4594.983,E2 4594.983} C_VEL
LIN {X 0,Y 523.501,Z 758.543,A -85,B 0,C 180,E1 4598.738,E2 4598.738} C_VEL
LIN {X 0,Y 523.983,Z 742.332,A -85,B 0,C 180,E1 4602.308,E2 4602.308} C_VEL
LIN {X 0,Y 524.845,Z 721.396,A -85,B 0,C 180,E1 4605.481,E2 4605.481} C_VEL
LIN {X 0,Y 525.866,Z 696.591,A -85,B 0,C 180,E1 4608.088,E2 4608.088} C_VEL
LIN {X 0,Y 527.077,Z 666.046,A -85,B 0,C 180,E1 4610.373,E2 4610.373} C_VEL
LIN {X 0,Y 528.202,Z 633.006,A -85,B 0,C 180,E1 4612.043,E2 4612.043} C_VEL
LIN {X 0,Y 528.873,Z 599.233,A -85,B 0,C 180,E1 4613.056,E2 4613.056} C_VEL
LIN {X 0,Y 528.331,Z 545.876,A -85,B 0,C 180,E1 4613.864,E2 4613.864} C_VEL
LIN {X 0,Y 522.719,Z 526.81,A -85,B 0,C 180,E1 4614.394,E2 4614.394} C_VEL
LIN {X 0,Y 522.356,Z 526.81,A -85,B 0,C 180,E1 4619.608,E2 4619.608} C_VEL
LIN {X 0,Y 522.3,Z 526.81,A -85,B 0,C 180,E1 4625.753,E2 4625.753} C_VEL
LIN {X 0,Y 522.406,Z 526.81,A -85,B 0,C 180,E1 4631.81,E2 4631.81} C_VEL
LIN {X 0,Y 522.322,Z 526.81,A -85,B 0,C 180,E1 4638.196,E2 4638.196} C_VEL
LIN {X 0,Y 522.321,Z 526.81,A -85,B 0,C 180,E1 4644.576,E2 4644.576} C_VEL
LIN {X 0,Y 522.428,Z 526.81,A -85,B 0,C 180,E1 4650.49,E2 4650.49} C_VEL
LIN {X 0,Y 522.489,Z 526.81,A -85,B 0,C 180,E1 4656.072,E2 4656.072} C_VEL
LIN {X 0,Y 522.617,Z 526.81,A -85,B 0,C 180,E1 4661.423,E2 4661.423} C_VEL
LIN {X 0,Y 522.708,Z 527.532,A -85,B 0,C 180,E1 4665.856,E2 4665.856} C_VEL
LIN {X 0,Y 525.605,Z 544.735,A -85,B 0,C 180,E1 4666.593,E2 4666.593} C_VEL
LIN {X 0,Y 525.041,Z 569.117,A -85,B 0,C 180,E1 4668.044,E2 4668.044} C_VEL
LIN {X 0,Y 524.424,Z 590.217,A -85,B 0,C 180,E1 4670.03,E2 4670.03} C_VEL
LIN {X 0,Y 523.878,Z 607.345,A -85,B 0,C 180,E1 4672.533,E2 4672.533} C_VEL
LIN {X 0,Y 523.589,Z 619.217,A -85,B 0,C 180,E1 4675.424,E2 4675.424} C_VEL
LIN {X 0,Y 523.404,Z 624.898,A -85,B 0,C 180,E1 4678.348,E2 4678.348} C_VEL
LIN {X 0,Y 523.423,Z 625.684,A -85,B 0,C 180,E1 4680.005,E2 4680.005} C_VEL
LIN {X 0,Y 523.45,Z 623.576,A -85,B 0,C 180,E1 4682.492,E2 4682.492} C_VEL
LIN {X 0,Y 523.618,Z 615.841,A -85,B 0,C 180,E1 4685.397,E2 4685.397} C_VEL
LIN {X 0,Y 523.866,Z 602.561,A -85,B 0,C 180,E1 4688.104,E2 4688.104} C_VEL
LIN {X 0,Y 524.427,Z 584.706,A -85,B 0,C 180,E1 4690.404,E2 4690.404} C_VEL
LIN {X 0,Y 525.056,Z 562.179,A -85,B 0,C 180,E1 4692.283,E2 4692.283} C_VEL
LIN {X 0,Y 524.859,Z 537.956,A -85,B 0,C 180,E1 4693.557,E2 4693.557} C_VEL
LIN {X 0,Y 522.612,Z 526.81,A -85,B 0,C 180,E1 4694.079,E2 4694.079} C_VEL
LIN {X 0,Y 522.622,Z 526.81,A -85,B 0,C 180,E1 4700.348,E2 4700.348} C_VEL
LIN {X 0,Y 522.431,Z 526.81,A -85,B 0,C 180,E1 4706.04,E2 4706.04} C_VEL
LIN {X 0,Y 522.362,Z 526.81,A -85,B 0,C 180,E1 4711.453,E2 4711.453} C_VEL
LIN {X 0,Y 522.268,Z 526.81,A -85,B 0,C 180,E1 4717.507,E2 4717.507} C_VEL
LIN {X 0,Y 522.328,Z 526.81,A -85,B 0,C 180,E1 4723.553,E2 4723.553} C_VEL
LIN {X 0,Y 522.384,Z 526.81,A -85,B 0,C 180,E1 4728.906,E2 4728.906} C_VEL
LIN {X 0,Y 522.328,Z 526.81,A -85,B 0,C 180,E1 4734.563,E2 4734.563} C_VEL
LIN {X 0,Y 522.404,Z 526.81,A -85,B 0,C 180,E1 4740.477,E2 4740.477} C_VEL
LIN {X 0,Y 522.57,Z 526.81,A -85,B 0,C 180,E1 4746.065,E2 4746.065} C_VEL
LIN {X 0,Y 522.725,Z 526.81,A -85,B 0,C 180,E1 4751.417,E2 4751.417} C_VEL
LIN {X 0,Y 522.629,Z 526.81,A -85,B 0,C 180,E1 4758.296,E2 4758.296} C_VEL
LIN {X 0,Y 522.939,Z 526.81,A -85,B 0,C 180,E1 4763.346,E2 4763.346} C_VEL
LIN {X 0,Y 522.943,Z 526.81,A -85,B 0,C 180,E1 4769.996,E2 4769.996} C_VEL
LIN {X 0,Y 522.876,Z 526.81,A -85,B 0,C 180,E1 4774.98,E2 4774.98} C_VEL
LIN {X 0,Y 522.781,Z 526.81,A -85,B 0,C 180,E1 4780.022,E2 4780.022} C_VEL
LIN {X 0,Y 522.695,Z 526.81,A -85,B 0,C 180,E1 4785.107,E2 4785.107} C_VEL
LIN {X 0,Y 522.621,Z 526.81,A -85,B 0,C 180,E1 4790.339,E2 4790.339} C_VEL
LIN {X 0,Y 522.428,Z 526.81,A -85,B 0,C 180,E1 4796.043,E2 4796.043} C_VEL
LIN {X 0,Y 522.353,Z 526.81,A -85,B 0,C 180,E1 4801.444,E2 4801.444} C_VEL
LIN {X 0,Y 522.26,Z 526.81,A -85,B 0,C 180,E1 4807.498,E2 4807.498} C_VEL
LIN {X 0,Y 522.291,Z 526.81,A -85,B 0,C 180,E1 4813.55,E2 4813.55} C_VEL
LIN {X 0,Y 522.407,Z 526.81,A -85,B 0,C 180,E1 4818.892,E2 4818.892} C_VEL
LIN {X 0,Y 522.313,Z 526.81,A -85,B 0,C 180,E1 4824.563,E2 4824.563} C_VEL
LIN {X 0,Y 522.385,Z 526.81,A -85,B 0,C 180,E1 4830.476,E2 4830.476} C_VEL
LIN {X 0,Y 522.557,Z 526.81,A -85,B 0,C 180,E1 4836.065,E2 4836.065} C_VEL
LIN {X 0,Y 522.742,Z 526.81,A -85,B 0,C 180,E1 4841.417,E2 4841.417} C_VEL
LIN {X 0,Y 522.634,Z 526.81,A -85,B 0,C 180,E1 4848.295,E2 4848.295} C_VEL
LIN {X 0,Y 522.915,Z 526.81,A -85,B 0,C 180,E1 4853.344,E2 4853.344} C_VEL
LIN {X 0,Y 522.918,Z 526.81,A -85,B 0,C 180,E1 4859.995,E2 4859.995} C_VEL
LIN {X 0,Y 522.851,Z 526.81,A -85,B 0,C 180,E1 4864.978,E2 4864.978} C_VEL
LIN {X 0,Y 522.722,Z 526.81,A -85,B 0,C 180,E1 4870.022,E2 4870.022} C_VEL
LIN {X 0,Y 522.654,Z 526.81,A -85,B 0,C 180,E1 4875.107,E2 4875.107} C_VEL
LIN {X 0,Y 522.584,Z 526.81,A -85,B 0,C 180,E1 4880.338,E2 4880.338} C_VEL
LIN {X 0,Y 522.432,Z 526.81,A -85,B 0,C 180,E1 4886.058,E2 4886.058} C_VEL
LIN {X 0,Y 522.408,Z 526.81,A -85,B 0,C 180,E1 4891.438,E2 4891.438} C_VEL
LIN {X 0,Y 522.482,Z 526.81,A -85,B 0,C 180,E1 4892.699,E2 4892.699} C_VEL
LIN {X 0,Y 520.037,Z 526.81,A -85,B 0,C 180,E1 4894.111,E2 4894.111} C_VEL
LIN {X 0,Y 514.557,Z 526.81,A -85,B 0,C 180,E1 4896.226,E2 4896.226} C_VEL
LIN {X 0,Y 514.451,Z 526.81,A -85,B 0,C 180,E1 4896.471,E2 4896.471} C_VEL
LIN {X 0,Y 514.289,Z 526.81,A -85,B 0,C 180,E1 4902.614,E2 4902.614} C_VEL
LIN {X 0,Y 514.264,Z 526.81,A -85,B 0,C 180,E1 4907.384,E2 4907.384} C_VEL
LIN {X 0,Y 514.298,Z 526.81,A -85,B 0,C 180,E1 4912.63,E2 4912.63} C_VEL
LIN {X 0,Y 514.434,Z 526.81,A -85,B 0,C 180,E1 4918.582,E2 4918.582} C_VEL
